LIN {X 0,Y 447.407,Z 741.258,A -85,B 0,C 180,E1 -8717.643,E2 -8717.643} C_VEL
LIN {X 0,Y 446.849,Z 749.798,A -85,B 0,C 180,E1 -8718.663,E2 -8718.663} C_VEL
LIN {X 0,Y 446.393,Z 757.677,A -85,B 0,C 180,E1 -8719.799,E2 -8719.799} C_VEL
LIN {X 0,Y 445.992,Z 765.376,A -85,B 0,C 180,E1 -8721.163,E2 -8721.163} C_VEL
LIN {X 0,Y 445.668,Z 772.472,A -85,B 0,C 180,E1 -8722.753,E2 -8722.753} C_VEL
LIN {X 0,Y 445.494,Z 776.598,A -85,B 0,C 180,E1 -8723.926,E2 -8723.926} C_VEL
LIN {X 0,Y 445.417,Z 780.807,A -85,B 0,C 180,E1 -8725.476,E2 -8725.476} C_VEL
LIN {X 0,Y 445.381,Z 782.67,A -85,B 0,C 180,E1 -8726.382,E2 -8726.382} C_VEL
LIN {X 0,Y 445.433,Z 784.067,A -85,B 0,C 180,E1 -8727.288,E2 -8727.288} C_VEL
LIN {X 0,Y 445.338,Z 785.666,A -85,B 0,C 180,E1 -8729.097,E2 -8729.097} C_VEL
LIN {X 0,Y 445.342,Z 785.882,A -85,B 0,C 180,E1 -8730.001,E2 -8730.001} C_VEL
LIN {X 0,Y 445.338,Z 785.664,A -85,B 0,C 180,E1 -8730.905,E2 -8730.905} C_VEL
LIN {X 0,Y 445.433,Z 784.061,A -85,B 0,C 180,E1 -8732.714,E2 -8732.714} C_VEL
LIN {X 0,Y 445.381,Z 782.661,A -85,B 0,C 180,E1 -8733.62,E2 -8733.62} C_VEL
LIN {X 0,Y 445.482,Z 779.728,A -85,B 0,C 180,E1 -8734.979,E2 -8734.979} C_VEL
LIN {X 0,Y 445.576,Z 774.321,A -85,B 0,C 180,E1 -8736.749,E2 -8736.749} C_VEL
LIN {X 0,Y 445.848,Z 768.627,A -85,B 0,C 180,E1 -8738.157,E2 -8738.157} C_VEL
LIN {X 0,Y 446.16,Z 761.722,A -85,B 0,C 180,E1 -8739.521,E2 -8739.521} C_VEL
LIN {X 0,Y 446.611,Z 753.085,A -85,B 0,C 180,E1 -8740.886,E2 -8740.886} C_VEL
LIN {X 0,Y 447.213,Z 744.233,A -85,B 0,C 180,E1 -8742.019,E2 -8742.019} C_VEL
LIN {X 0,Y 447.682,Z 735.24,A -85,B 0,C 180,E1 -8742.972,E2 -8742.972} C_VEL
LIN {X 0,Y 448.293,Z 723.879,A -85,B 0,C 180,E1 -8743.949,E2 -8743.949} C_VEL
LIN {X 0,Y 448.894,Z 712.012,A -85,B 0,C 180,E1 -8744.74,E2 -8744.74} C_VEL
LIN {X 0,Y 449.496,Z 699.666,A -85,B 0,C 180,E1 -8745.357,E2 -8745.357} C_VEL
LIN {X 0,Y 449.946,Z 686.98,A -85,B 0,C 180,E1 -8745.806,E2 -8745.806} C_VEL
LIN {X 0,Y 450.236,Z 673.706,A -85,B 0,C 180,E1 -8746.086,E2 -8746.086} C_VEL
LIN {X 0,Y 450.721,Z 593.513,A -85,B 0,C 180,E1 -8747.374,E2 -8747.374} C_VEL
LIN {X 0,Y 447.503,Z 573.501,A -85,B 0,C 180,E1 -8747.859,E2 -8747.859} C_VEL
LIN {X 0,Y 448.187,Z 559.557,A -85,B 0,C 180,E1 -8750.421,E2 -8750.421} C_VEL
LIN {X 0,Y 449.049,Z 544.405,A -85,B 0,C 180,E1 -8753.278,E2 -8753.278} C_VEL
LIN {X 0,Y 448.611,Z 539.586,A -85,B 0,C 180,E1 -8754.233,E2 -8754.233} C_VEL
LIN {X 0,Y 446.536,Z 529.051,A -85,B 0,C 180,E1 -8756.444,E2 -8756.444} C_VEL
LIN {X 0,Y 446.452,Z 528.852,A -85,B 0,C 180,E1 -8759.21,E2 -8759.21} C_VEL
LIN {X 0,Y 446.426,Z 528.878,A -85,B 0,C 180,E1 -8762.362,E2 -8762.362} C_VEL
LIN {X 0,Y 446.423,Z 528.875,A -85,B 0,C 180,E1 -8765.626,E2 -8765.626} C_VEL
LIN {X 0,Y 446.448,Z 528.87,A -85,B 0,C 180,E1 -8769.027,E2 -8769.027} C_VEL
LIN {X 0,Y 446.439,Z 528.875,A -85,B 0,C 180,E1 -8772.278,E2 -8772.278} C_VEL
LIN {X 0,Y 446.458,Z 528.871,A -85,B 0,C 180,E1 -8775.104,E2 -8775.104} C_VEL
LIN {X 0,Y 446.432,Z 528.875,A -85,B 0,C 180,E1 -8778.609,E2 -8778.609} C_VEL
LIN {X 0,Y 446.449,Z 528.871,A -85,B 0,C 180,E1 -8780.973,E2 -8780.973} C_VEL
LIN {X 0,Y 446.426,Z 528.877,A -85,B 0,C 180,E1 -8784.374,E2 -8784.374} C_VEL
LIN {X 0,Y 446.426,Z 528.879,A -85,B 0,C 180,E1 -8787.639,E2 -8787.639} C_VEL
LIN {X 0,Y 446.49,Z 528.871,A -85,B 0,C 180,E1 -8791.309,E2 -8791.309} C_VEL
LIN {X 0,Y 446.544,Z 529.135,A -85,B 0,C 180,E1 -8791.774,E2 -8791.774} C_VEL
LIN {X 0,Y 448.876,Z 539.427,A -85,B 0,C 180,E1 -8793.454,E2 -8793.454} C_VEL
LIN {X 0,Y 449.618,Z 544.795,A -85,B 0,C 180,E1 -8794.293,E2 -8794.293} C_VEL
LIN {X 0,Y 448.993,Z 565.446,A -85,B 0,C 180,E1 -8797.299,E2 -8797.299} C_VEL
LIN {X 0,Y 448.285,Z 587.456,A -85,B 0,C 180,E1 -8800.545,E2 -8800.545} C_VEL
LIN {X 0,Y 447.587,Z 611.18,A -85,B 0,C 180,E1 -8804.051,E2 -8804.051} C_VEL
LIN {X 0,Y 446.999,Z 631.561,A -85,B 0,C 180,E1 -8807.047,E2 -8807.047} C_VEL
LIN {X 0,Y 448.391,Z 644.528,A -85,B 0,C 180,E1 -8807.365,E2 -8807.365} C_VEL
LIN {X 0,Y 447.727,Z 703.384,A -85,B 0,C 180,E1 -8808.484,E2 -8808.484} C_VEL
LIN {X 0,Y 447.557,Z 713.56,A -85,B 0,C 180,E1 -8808.823,E2 -8808.823} C_VEL
LIN {X 0,Y 447.25,Z 724.586,A -85,B 0,C 180,E1 -8809.36,E2 -8809.36} C_VEL
LIN {X 0,Y 446.948,Z 734.395,A -85,B 0,C 180,E1 -8810.04,E2 -8810.04} C_VEL
LIN {X 0,Y 446.644,Z 742.148,A -85,B 0,C 180,E1 -8810.719,E2 -8810.719} C_VEL
LIN {X 0,Y 446.274,Z 750.496,A -85,B 0,C 180,E1 -8811.624,E2 -8811.624} C_VEL
LIN {X 0,Y 445.989,Z 758.487,A -85,B 0,C 180,E1 -8812.758,E2 -8812.758} C_VEL
LIN {X 0,Y 445.802,Z 763.618,A -85,B 0,C 180,E1 -8813.664,E2 -8813.664} C_VEL
LIN {X 0,Y 445.686,Z 767.819,A -85,B 0,C 180,E1 -8814.571,E2 -8814.571} C_VEL
LIN {X 0,Y 445.501,Z 771.222,A -85,B 0,C 180,E1 -8815.476,E2 -8815.476} C_VEL
LIN {X 0,Y 445.504,Z 773.912,A -85,B 0,C 180,E1 -8816.382,E2 -8816.382} C_VEL
LIN {X 0,Y 445.455,Z 775.959,A -85,B 0,C 180,E1 -8817.287,E2 -8817.287} C_VEL
LIN {X 0,Y 445.357,Z 777.408,A -85,B 0,C 180,E1 -8818.191,E2 -8818.191} C_VEL
LIN {X 0,Y 445.314,Z 778.286,A -85,B 0,C 180,E1 -8819.096,E2 -8819.096} C_VEL
LIN {X 0,Y 445.315,Z 778.58,A -85,B 0,C 180,E1 -8820,E2 -8820} C_VEL
LIN {X 0,Y 445.315,Z 778.281,A -85,B 0,C 180,E1 -8820.904,E2 -8820.904} C_VEL
LIN {X 0,Y 445.357,Z 777.404,A -85,B 0,C 180,E1 -8821.809,E2 -8821.809} C_VEL
LIN {X 0,Y 445.488,Z 775.061,A -85,B 0,C 180,E1 -8823.165,E2 -8823.165} C_VEL
LIN {X 0,Y 445.477,Z 772.717,A -85,B 0,C 180,E1 -8824.071,E2 -8824.071} C_VEL
LIN {X 0,Y 445.56,Z 769.687,A -85,B 0,C 180,E1 -8824.977,E2 -8824.977} C_VEL
LIN {X 0,Y 445.736,Z 764.784,A -85,B 0,C 180,E1 -8826.11,E2 -8826.11} C_VEL
LIN {X 0,Y 445.92,Z 760.093,A -85,B 0,C 180,E1 -8826.983,E2 -8826.983} C_VEL
LIN {X 0,Y 446.07,Z 753.905,A -85,B 0,C 180,E1 -8827.924,E2 -8827.924} C_VEL
LIN {X 0,Y 446.349,Z 746.57,A -85,B 0,C 180,E1 -8828.831,E2 -8828.831} C_VEL
LIN {X 0,Y 446.748,Z 737.266,A -85,B 0,C 180,E1 -8829.736,E2 -8829.736} C_VEL
LIN {X 0,Y 447.058,Z 728.149,A -85,B 0,C 180,E1 -8830.416,E2 -8830.416} C_VEL
LIN {X 0,Y 447.317,Z 718.258,A -85,B 0,C 180,E1 -8830.982,E2 -8830.982} C_VEL
LIN {X 0,Y 447.568,Z 707.509,A -85,B 0,C 180,E1 -8831.406,E2 -8831.406} C_VEL
LIN {X 0,Y 447.655,Z 697.084,A -85,B 0,C 180,E1 -8831.662,E2 -8831.662} C_VEL
LIN {X 0,Y 448.07,Z 642.126,A -85,B 0,C 180,E1 -8832.648,E2 -8832.648} C_VEL
LIN {X 0,Y 446.85,Z 631.601,A -85,B 0,C 180,E1 -8832.889,E2 -8832.889} C_VEL
LIN {X 0,Y 447.122,Z 621.716,A -85,B 0,C 180,E1 -8834.333,E2 -8834.333} C_VEL
LIN {X 0,Y 447.779,Z 600.173,A -85,B 0,C 180,E1 -8837.586,E2 -8837.586} C_VEL
LIN {X 0,Y 448.48,Z 579.967,A -85,B 0,C 180,E1 -8840.646,E2 -8840.646} C_VEL
LIN {X 0,Y 449.352,Z 556.333,A -85,B 0,C 180,E1 -8844.24,E2 -8844.24} C_VEL
LIN {X 0,Y 449.698,Z 545.085,A -85,B 0,C 180,E1 -8845.95,E2 -8845.95} C_VEL
LIN {X 0,Y 447.465,Z 533.4,A -85,B 0,C 180,E1 -8847.857,E2 -8847.857} C_VEL
LIN {X 0,Y 446.517,Z 528.97,A -85,B 0,C 180,E1 -8848.636,E2 -8848.636} C_VEL
LIN {X 0,Y 446.426,Z 528.879,A -85,B 0,C 180,E1 -8852.361,E2 -8852.361} C_VEL
LIN {X 0,Y 446.426,Z 528.874,A -85,B 0,C 180,E1 -8855.626,E2 -8855.626} C_VEL
LIN {X 0,Y 446.45,Z 528.869,A -85,B 0,C 180,E1 -8859.027,E2 -8859.027} C_VEL
LIN {X 0,Y 446.438,Z 528.854,A -85,B 0,C 180,E1 -8862.277,E2 -8862.277} C_VEL
LIN {X 0,Y 446.46,Z 528.867,A -85,B 0,C 180,E1 -8865.103,E2 -8865.103} C_VEL
LIN {X 0,Y 446.434,Z 528.869,A -85,B 0,C 180,E1 -8868.609,E2 -8868.609} C_VEL
LIN {X 0,Y 446.446,Z 528.861,A -85,B 0,C 180,E1 -8870.973,E2 -8870.973} C_VEL
LIN {X 0,Y 446.424,Z 528.878,A -85,B 0,C 180,E1 -8874.374,E2 -8874.374} C_VEL
LIN {X 0,Y 446.427,Z 528.873,A -85,B 0,C 180,E1 -8877.638,E2 -8877.638} C_VEL
LIN {X 0,Y 446.453,Z 528.873,A -85,B 0,C 180,E1 -8880.79,E2 -8880.79} C_VEL
LIN {X 0,Y 446.483,Z 528.867,A -85,B 0,C 180,E1 -8883.848,E2 -8883.848} C_VEL
LIN {X 0,Y 446.462,Z 528.879,A -85,B 0,C 180,E1 -8887.314,E2 -8887.314} C_VEL
LIN {X 0,Y 446.546,Z 529.43,A -85,B 0,C 180,E1 -8887.563,E2 -8887.563} C_VEL
LIN {X 0,Y 448.137,Z 537.779,A -85,B 0,C 180,E1 -8889.577,E2 -8889.577} C_VEL
LIN {X 0,Y 447.892,Z 544.522,A -85,B 0,C 180,E1 -8891.086,E2 -8891.086} C_VEL
LIN {X 0,Y 447.633,Z 546.914,A -85,B 0,C 180,E1 -8891.469,E2 -8891.469} C_VEL
LIN {X 0,Y 446.932,Z 551.667,A -85,B 0,C 180,E1 -8891.892,E2 -8891.892} C_VEL
LIN {X 0,Y 446.062,Z 557.135,A -85,B 0,C 180,E1 -8892.159,E2 -8892.159} C_VEL
LIN {X 0,Y 444.882,Z 565.287,A -85,B 0,C 180,E1 -8892.361,E2 -8892.361} C_VEL
LIN {X 0,Y 444.177,Z 573.6,A -85,B 0,C 180,E1 -8892.485,E2 -8892.485} C_VEL
LIN {X 0,Y 443.385,Z 657.161,A -85,B 0,C 180,E1 -8893.865,E2 -8893.865} C_VEL
LIN {X 0,Y 443.004,Z 671.025,A -85,B 0,C 180,E1 -8894.294,E2 -8894.294} C_VEL
LIN {X 0,Y 442.518,Z 683.422,A -85,B 0,C 180,E1 -8894.866,E2 -8894.866} C_VEL
LIN {X 0,Y 441.942,Z 695.268,A -85,B 0,C 180,E1 -8895.612,E2 -8895.612} C_VEL
LIN {X 0,Y 441.388,Z 706.67,A -85,B 0,C 180,E1 -8896.537,E2 -8896.537} C_VEL
LIN {X 0,Y 440.763,Z 716.867,A -85,B 0,C 180,E1 -8897.569,E2 -8897.569} C_VEL
LIN {X 0,Y 440.147,Z 726.052,A -85,B 0,C 180,E1 -8898.719,E2 -8898.719} C_VEL
LIN {X 0,Y 439.552,Z 734.97,A -85,B 0,C 180,E1 -8900.102,E2 -8900.102} C_VEL
LIN {X 0,Y 439.104,Z 742.146,A -85,B 0,C 180,E1 -8901.485,E2 -8901.485} C_VEL
LIN {X 0,Y 438.788,Z 746.99,A -85,B 0,C 180,E1 -8902.637,E2 -8902.637} C_VEL
LIN {X 0,Y 438.686,Z 751.69,A -85,B 0,C 180,E1 -8904.022,E2 -8904.022} C_VEL
LIN {X 0,Y 438.424,Z 755.29,A -85,B 0,C 180,E1 -8905.402,E2 -8905.402} C_VEL
LIN {X 0,Y 438.428,Z 757.148,A -85,B 0,C 180,E1 -8906.323,E2 -8906.323} C_VEL
LIN {X 0,Y 438.395,Z 758.551,A -85,B 0,C 180,E1 -8907.243,E2 -8907.243} C_VEL
LIN {X 0,Y 438.255,Z 760.167,A -85,B 0,C 180,E1 -8909.08,E2 -8909.08} C_VEL
LIN {X 0,Y 438.254,Z 760.402,A -85,B 0,C 180,E1 -8909.999,E2 -8909.999} C_VEL
LIN {X 0,Y 438.255,Z 760.216,A -85,B 0,C 180,E1 -8910.918,E2 -8910.918} C_VEL
LIN {X 0,Y 438.392,Z 758.667,A -85,B 0,C 180,E1 -8912.756,E2 -8912.756} C_VEL
LIN {X 0,Y 438.413,Z 757.314,A -85,B 0,C 180,E1 -8913.676,E2 -8913.676} C_VEL
LIN {X 0,Y 438.481,Z 754.45,A -85,B 0,C 180,E1 -8915.057,E2 -8915.057} C_VEL
LIN {X 0,Y 438.693,Z 750.563,A -85,B 0,C 180,E1 -8916.438,E2 -8916.438} C_VEL
LIN {X 0,Y 438.902,Z 745.555,A -85,B 0,C 180,E1 -8917.822,E2 -8917.822} C_VEL
LIN {X 0,Y 439.321,Z 739.248,A -85,B 0,C 180,E1 -8919.204,E2 -8919.204} C_VEL
LIN {X 0,Y 439.803,Z 731.349,A -85,B 0,C 180,E1 -8920.588,E2 -8920.588} C_VEL
LIN {X 0,Y 440.285,Z 723.299,A -85,B 0,C 180,E1 -8921.742,E2 -8921.742} C_VEL
LIN {X 0,Y 441.015,Z 713.467,A -85,B 0,C 180,E1 -8922.89,E2 -8922.89} C_VEL
LIN {X 0,Y 441.544,Z 702.694,A -85,B 0,C 180,E1 -8923.907,E2 -8923.907} C_VEL
LIN {X 0,Y 442.142,Z 691.584,A -85,B 0,C 180,E1 -8924.733,E2 -8924.733} C_VEL
LIN {X 0,Y 442.72,Z 679.605,A -85,B 0,C 180,E1 -8925.419,E2 -8925.419} C_VEL
LIN {X 0,Y 443.147,Z 666.472,A -85,B 0,C 180,E1 -8925.965,E2 -8925.965} C_VEL
LIN {X 0,Y 443.508,Z 653.263,A -85,B 0,C 180,E1 -8926.306,E2 -8926.306} C_VEL
LIN {X 0,Y 444.113,Z 567.024,A -85,B 0,C 180,E1 -8927.72,E2 -8927.72} C_VEL
LIN {X 0,Y 440.768,Z 550.156,A -85,B 0,C 180,E1 -8928.171,E2 -8928.171} C_VEL
LIN {X 0,Y 440.78,Z 547.921,A -85,B 0,C 180,E1 -8928.595,E2 -8928.595} C_VEL
LIN {X 0,Y 441.2,Z 539.437,A -85,B 0,C 180,E1 -8930.513,E2 -8930.513} C_VEL
LIN {X 0,Y 439.437,Z 529.822,A -85,B 0,C 180,E1 -8932.912,E2 -8932.912} C_VEL
LIN {X 0,Y 439.433,Z 529.742,A -85,B 0,C 180,E1 -8936.41,E2 -8936.41} C_VEL
LIN {X 0,Y 439.416,Z 529.744,A -85,B 0,C 180,E1 -8938.672,E2 -8938.672} C_VEL
LIN {X 0,Y 439.369,Z 529.753,A -85,B 0,C 180,E1 -8942.03,E2 -8942.03} C_VEL
LIN {X 0,Y 439.394,Z 529.752,A -85,B 0,C 180,E1 -8945.34,E2 -8945.34} C_VEL
LIN {X 0,Y 439.387,Z 529.75,A -85,B 0,C 180,E1 -8948.593,E2 -8948.593} C_VEL
LIN {X 0,Y 439.386,Z 529.751,A -85,B 0,C 180,E1 -8951.256,E2 -8951.256} C_VEL
LIN {X 0,Y 439.401,Z 529.741,A -85,B 0,C 180,E1 -8954.728,E2 -8954.728} C_VEL
LIN {X 0,Y 439.392,Z 529.752,A -85,B 0,C 180,E1 -8957.795,E2 -8957.795} C_VEL
LIN {X 0,Y 439.447,Z 529.734,A -85,B 0,C 180,E1 -8960.229,E2 -8960.229} C_VEL
LIN {X 0,Y 439.373,Z 529.756,A -85,B 0,C 180,E1 -8963.712,E2 -8963.712} C_VEL
LIN {X 0,Y 439.367,Z 529.754,A -85,B 0,C 180,E1 -8967.053,E2 -8967.053} C_VEL
LIN {X 0,Y 439.39,Z 529.749,A -85,B 0,C 180,E1 -8970.275,E2 -8970.275} C_VEL
LIN {X 0,Y 439.427,Z 529.748,A -85,B 0,C 180,E1 -8973.588,E2 -8973.588} C_VEL
LIN {X 0,Y 439.38,Z 529.748,A -85,B 0,C 180,E1 -8976.429,E2 -8976.429} C_VEL
LIN {X 0,Y 439.382,Z 529.752,A -85,B 0,C 180,E1 -8979.397,E2 -8979.397} C_VEL
LIN {X 0,Y 439.424,Z 529.741,A -85,B 0,C 180,E1 -8982.309,E2 -8982.309} C_VEL
LIN {X 0,Y 439.44,Z 529.741,A -85,B 0,C 180,E1 -8985.174,E2 -8985.174} C_VEL
LIN {X 0,Y 439.476,Z 529.738,A -85,B 0,C 180,E1 -8988.001,E2 -8988.001} C_VEL
LIN {X 0,Y 439.54,Z 529.734,A -85,B 0,C 180,E1 -8991.726,E2 -8991.726} C_VEL
LIN {X 0,Y 439.614,Z 529.72,A -85,B 0,C 180,E1 -8994.496,E2 -8994.496} C_VEL
LIN {X 0,Y 439.628,Z 529.718,A -85,B 0,C 180,E1 -8998.168,E2 -8998.168} C_VEL
LIN {X 0,Y 439.757,Z 529.706,A -85,B 0,C 180,E1 -9000,E2 -9000} C_VEL
LIN {X 0,Y 439.649,Z 529.712,A -85,B 0,C 180,E1 -9002.749,E2 -9002.749} C_VEL
LIN {X 0,Y 439.61,Z 529.721,A -85,B 0,C 180,E1 -9006.425,E2 -9006.425} C_VEL
LIN {X 0,Y 439.493,Z 529.737,A -85,B 0,C 180,E1 -9009.202,E2 -9009.202} C_VEL
LIN {X 0,Y 439.496,Z 529.735,A -85,B 0,C 180,E1 -9012.727,E2 -9012.727} C_VEL
LIN {X 0,Y 439.44,Z 529.737,A -85,B 0,C 180,E1 -9016.349,E2 -9016.349} C_VEL
LIN {X 0,Y 439.423,Z 529.751,A -85,B 0,C 180,E1 -9019.625,E2 -9019.625} C_VEL
LIN {X 0,Y 439.358,Z 529.75,A -85,B 0,C 180,E1 -9022.576,E2 -9022.576} C_VEL
LIN {X 0,Y 439.399,Z 529.752,A -85,B 0,C 180,E1 -9025.585,E2 -9025.585} C_VEL
LIN {X 0,Y 439.411,Z 529.747,A -85,B 0,C 180,E1 -9028.674,E2 -9028.674} C_VEL
LIN {X 0,Y 439.375,Z 529.754,A -85,B 0,C 180,E1 -9032.034,E2 -9032.034} C_VEL
LIN {X 0,Y 439.39,Z 529.748,A -85,B 0,C 180,E1 -9035.342,E2 -9035.342} C_VEL
LIN {X 0,Y 439.385,Z 529.749,A -85,B 0,C 180,E1 -9038.595,E2 -9038.595} C_VEL
LIN {X 0,Y 439.383,Z 529.752,A -85,B 0,C 180,E1 -9041.258,E2 -9041.258} C_VEL
LIN {X 0,Y 439.4,Z 529.748,A -85,B 0,C 180,E1 -9044.73,E2 -9044.73} C_VEL
LIN {X 0,Y 439.408,Z 529.749,A -85,B 0,C 180,E1 -9047.799,E2 -9047.799} C_VEL
LIN {X 0,Y 439.447,Z 529.739,A -85,B 0,C 180,E1 -9050.231,E2 -9050.231} C_VEL
LIN {X 0,Y 439.374,Z 529.748,A -85,B 0,C 180,E1 -9053.714,E2 -9053.714} C_VEL
LIN {X 0,Y 439.37,Z 529.733,A -85,B 0,C 180,E1 -9057.055,E2 -9057.055} C_VEL
LIN {X 0,Y 439.38,Z 529.723,A -85,B 0,C 180,E1 -9060.275,E2 -9060.275} C_VEL
LIN {X 0,Y 439.469,Z 529.836,A -85,B 0,C 180,E1 -9063.272,E2 -9063.272} C_VEL
LIN {X 0,Y 441.813,Z 541.718,A -85,B 0,C 180,E1 -9065.821,E2 -9065.821} C_VEL
LIN {X 0,Y 442.142,Z 545.523,A -85,B 0,C 180,E1 -9066.586,E2 -9066.586} C_VEL
LIN {X 0,Y 441.101,Z 562.606,A -85,B 0,C 180,E1 -9069.856,E2 -9069.856} C_VEL
LIN {X 0,Y 440.59,Z 573.22,A -85,B 0,C 180,E1 -9071.841,E2 -9071.841} C_VEL
LIN {X 0,Y 442.189,Z 582.98,A -85,B 0,C 180,E1 -9072.105,E2 -9072.105} C_VEL
LIN {X 0,Y 444.109,Z 596.392,A -85,B 0,C 180,E1 -9072.407,E2 -9072.407} C_VEL
LIN {X 0,Y 443.294,Z 681.341,A -85,B 0,C 180,E1 -9073.805,E2 -9073.805} C_VEL
LIN {X 0,Y 442.826,Z 694.585,A -85,B 0,C 180,E1 -9074.201,E2 -9074.201} C_VEL
LIN {X 0,Y 442.286,Z 707.863,A -85,B 0,C 180,E1 -9074.801,E2 -9074.801} C_VEL
LIN {X 0,Y 441.659,Z 719.016,A -85,B 0,C 180,E1 -9075.486,E2 -9075.486} C_VEL
LIN {X 0,Y 441.048,Z 729.687,A -85,B 0,C 180,E1 -9076.323,E2 -9076.323} C_VEL
LIN {X 0,Y 440.443,Z 741.055,A -85,B 0,C 180,E1 -9077.444,E2 -9077.444} C_VEL
LIN {X 0,Y 439.873,Z 749.594,A -85,B 0,C 180,E1 -9078.481,E2 -9078.481} C_VEL
LIN {X 0,Y 439.371,Z 757.473,A -85,B 0,C 180,E1 -9079.634,E2 -9079.634} C_VEL
LIN {X 0,Y 438.937,Z 765.171,A -85,B 0,C 180,E1 -9081.02,E2 -9081.02} C_VEL
LIN {X 0,Y 438.606,Z 772.267,A -85,B 0,C 180,E1 -9082.636,E2 -9082.636} C_VEL
LIN {X 0,Y 438.393,Z 776.825,A -85,B 0,C 180,E1 -9083.967,E2 -9083.967} C_VEL
LIN {X 0,Y 438.346,Z 780.603,A -85,B 0,C 180,E1 -9085.403,E2 -9085.403} C_VEL
LIN {X 0,Y 438.283,Z 782.465,A -85,B 0,C 180,E1 -9086.323,E2 -9086.323} C_VEL
LIN {X 0,Y 438.341,Z 783.863,A -85,B 0,C 180,E1 -9087.244,E2 -9087.244} C_VEL
LIN {X 0,Y 438.252,Z 785.462,A -85,B 0,C 180,E1 -9089.082,E2 -9089.082} C_VEL
LIN {X 0,Y 438.253,Z 785.678,A -85,B 0,C 180,E1 -9090.001,E2 -9090.001} C_VEL
LIN {X 0,Y 438.278,Z 784.851,A -85,B 0,C 180,E1 -9091.839,E2 -9091.839} C_VEL
LIN {X 0,Y 438.341,Z 783.856,A -85,B 0,C 180,E1 -9092.758,E2 -9092.758} C_VEL
LIN {X 0,Y 438.283,Z 782.456,A -85,B 0,C 180,E1 -9093.678,E2 -9093.678} C_VEL
LIN {X 0,Y 438.392,Z 779.522,A -85,B 0,C 180,E1 -9095.059,E2 -9095.059} C_VEL
LIN {X 0,Y 438.449,Z 775.547,A -85,B 0,C 180,E1 -9096.443,E2 -9096.443} C_VEL
LIN {X 0,Y 438.724,Z 769.432,A -85,B 0,C 180,E1 -9098.058,E2 -9098.058} C_VEL
LIN {X 0,Y 439.066,Z 762.753,A -85,B 0,C 180,E1 -9099.444,E2 -9099.444} C_VEL
LIN {X 0,Y 439.523,Z 754.466,A -85,B 0,C 180,E1 -9100.83,E2 -9100.83} C_VEL
LIN {X 0,Y 440.111,Z 745.976,A -85,B 0,C 180,E1 -9101.982,E2 -9101.982} C_VEL
LIN {X 0,Y 440.68,Z 735.869,A -85,B 0,C 180,E1 -9103.098,E2 -9103.098} C_VEL
LIN {X 0,Y 441.296,Z 725.1,A -85,B 0,C 180,E1 -9104.057,E2 -9104.057} C_VEL
LIN {X 0,Y 441.923,Z 713.727,A -85,B 0,C 180,E1 -9104.86,E2 -9104.86} C_VEL
LIN {X 0,Y 442.547,Z 702.06,A -85,B 0,C 180,E1 -9105.486,E2 -9105.486} C_VEL
LIN {X 0,Y 443.011,Z 689.516,A -85,B 0,C 180,E1 -9105.971,E2 -9105.971} C_VEL
LIN {X 0,Y 443.385,Z 676.797,A -85,B 0,C 180,E1 -9106.282,E2 -9106.282} C_VEL
LIN {X 0,Y 443.999,Z 594.924,A -85,B 0,C 180,E1 -9107.619,E2 -9107.619} C_VEL
LIN {X 0,Y 440.562,Z 573.533,A -85,B 0,C 180,E1 -9108.133,E2 -9108.133} C_VEL
LIN {X 0,Y 440.689,Z 570.679,A -85,B 0,C 180,E1 -9108.6,E2 -9108.6} C_VEL
LIN {X 0,Y 441.86,Z 550.549,A -85,B 0,C 180,E1 -9112.442,E2 -9112.442} C_VEL
LIN {X 0,Y 442.138,Z 544.222,A -85,B 0,C 180,E1 -9113.664,E2 -9113.664} C_VEL
LIN {X 0,Y 440.34,Z 534.062,A -85,B 0,C 180,E1 -9115.777,E2 -9115.777} C_VEL
LIN {X 0,Y 439.475,Z 529.804,A -85,B 0,C 180,E1 -9116.746,E2 -9116.746} C_VEL
LIN {X 0,Y 439.385,Z 529.736,A -85,B 0,C 180,E1 -9119.726,E2 -9119.726} C_VEL
LIN {X 0,Y 439.376,Z 529.754,A -85,B 0,C 180,E1 -9122.946,E2 -9122.946} C_VEL
LIN {X 0,Y 439.378,Z 529.756,A -85,B 0,C 180,E1 -9126.288,E2 -9126.288} C_VEL
LIN {X 0,Y 439.405,Z 529.753,A -85,B 0,C 180,E1 -9129.849,E2 -9129.849} C_VEL
LIN {X 0,Y 439.386,Z 529.752,A -85,B 0,C 180,E1 -9132.627,E2 -9132.627} C_VEL
LIN {X 0,Y 439.405,Z 529.75,A -85,B 0,C 180,E1 -9135.271,E2 -9135.271} C_VEL
LIN {X 0,Y 439.392,Z 529.752,A -85,B 0,C 180,E1 -9138.743,E2 -9138.743} C_VEL
LIN {X 0,Y 439.386,Z 529.755,A -85,B 0,C 180,E1 -9141.607,E2 -9141.607} C_VEL
LIN {X 0,Y 439.405,Z 529.749,A -85,B 0,C 180,E1 -9144.844,E2 -9144.844} C_VEL
LIN {X 0,Y 439.377,Z 529.758,A -85,B 0,C 180,E1 -9148.14,E2 -9148.14} C_VEL
LIN {X 0,Y 439.479,Z 529.934,A -85,B 0,C 180,E1 -9151.397,E2 -9151.397} C_VEL
LIN {X 0,Y 442.015,Z 540.745,A -85,B 0,C 180,E1 -9153.218,E2 -9153.218} C_VEL
LIN {X 0,Y 442.837,Z 546.431,A -85,B 0,C 180,E1 -9154.123,E2 -9154.123} C_VEL
LIN {X 0,Y 442.172,Z 565.852,A -85,B 0,C 180,E1 -9156.992,E2 -9156.992} C_VEL
LIN {X 0,Y 441.413,Z 587.891,A -85,B 0,C 180,E1 -9160.283,E2 -9160.283} C_VEL
LIN {X 0,Y 440.69,Z 611.421,A -85,B 0,C 180,E1 -9163.794,E2 -9163.794} C_VEL
LIN {X 0,Y 440.074,Z 631.467,A -85,B 0,C 180,E1 -9166.782,E2 -9166.782} C_VEL
LIN {X 0,Y 441.551,Z 645.299,A -85,B 0,C 180,E1 -9167.145,E2 -9167.145} C_VEL
LIN {X 0,Y 440.795,Z 704.212,A -85,B 0,C 180,E1 -9168.3,E2 -9168.3} C_VEL
LIN {X 0,Y 440.605,Z 713.419,A -85,B 0,C 180,E1 -9168.616,E2 -9168.616} C_VEL
LIN {X 0,Y 440.309,Z 723.945,A -85,B 0,C 180,E1 -9169.132,E2 -9169.132} C_VEL
LIN {X 0,Y 439.986,Z 733.226,A -85,B 0,C 180,E1 -9169.764,E2 -9169.764} C_VEL
LIN {X 0,Y 439.677,Z 741.161,A -85,B 0,C 180,E1 -9170.454,E2 -9170.454} C_VEL
LIN {X 0,Y 439.334,Z 748.677,A -85,B 0,C 180,E1 -9171.259,E2 -9171.259} C_VEL
LIN {X 0,Y 439.039,Z 755.676,A -85,B 0,C 180,E1 -9172.18,E2 -9172.18} C_VEL
LIN {X 0,Y 438.831,Z 761.873,A -85,B 0,C 180,E1 -9173.194,E2 -9173.194} C_VEL
LIN {X 0,Y 438.731,Z 766.011,A -85,B 0,C 180,E1 -9174.023,E2 -9174.023} C_VEL
LIN {X 0,Y 438.517,Z 769.796,A -85,B 0,C 180,E1 -9174.943,E2 -9174.943} C_VEL
LIN {X 0,Y 438.435,Z 772.823,A -85,B 0,C 180,E1 -9175.863,E2 -9175.863} C_VEL
LIN {X 0,Y 438.388,Z 776.047,A -85,B 0,C 180,E1 -9177.243,E2 -9177.243} C_VEL
LIN {X 0,Y 438.28,Z 777.486,A -85,B 0,C 180,E1 -9178.162,E2 -9178.162} C_VEL
LIN {X 0,Y 438.229,Z 778.351,A -85,B 0,C 180,E1 -9179.081,E2 -9179.081} C_VEL
LIN {X 0,Y 438.227,Z 778.636,A -85,B 0,C 180,E1 -9180,E2 -9180} C_VEL
LIN {X 0,Y 438.23,Z 778.324,A -85,B 0,C 180,E1 -9180.919,E2 -9180.919} C_VEL
LIN {X 0,Y 438.28,Z 777.425,A -85,B 0,C 180,E1 -9181.838,E2 -9181.838} C_VEL
LIN {X 0,Y 438.415,Z 775.03,A -85,B 0,C 180,E1 -9183.216,E2 -9183.216} C_VEL
LIN {X 0,Y 438.413,Z 771.156,A -85,B 0,C 180,E1 -9184.597,E2 -9184.597} C_VEL
LIN {X 0,Y 438.566,Z 767.72,A -85,B 0,C 180,E1 -9185.518,E2 -9185.518} C_VEL
LIN {X 0,Y 438.729,Z 762.194,A -85,B 0,C 180,E1 -9186.693,E2 -9186.693} C_VEL
LIN {X 0,Y 438.954,Z 755.305,A -85,B 0,C 180,E1 -9187.822,E2 -9187.822} C_VEL
LIN {X 0,Y 439.244,Z 748.216,A -85,B 0,C 180,E1 -9188.743,E2 -9188.743} C_VEL
LIN {X 0,Y 439.644,Z 739.42,A -85,B 0,C 180,E1 -9189.663,E2 -9189.663} C_VEL
LIN {X 0,Y 439.996,Z 729.246,A -85,B 0,C 180,E1 -9190.468,E2 -9190.468} C_VEL
LIN {X 0,Y 440.26,Z 719.62,A -85,B 0,C 180,E1 -9191.044,E2 -9191.044} C_VEL
LIN {X 0,Y 440.558,Z 708.014,A -85,B 0,C 180,E1 -9191.531,E2 -9191.531} C_VEL
LIN {X 0,Y 440.661,Z 696.322,A -85,B 0,C 180,E1 -9191.82,E2 -9191.82} C_VEL
LIN {X 0,Y 441.144,Z 643.139,A -85,B 0,C 180,E1 -9192.802,E2 -9192.802} C_VEL
LIN {X 0,Y 439.846,Z 631.675,A -85,B 0,C 180,E1 -9193.069,E2 -9193.069} C_VEL
LIN {X 0,Y 439.905,Z 627.77,A -85,B 0,C 180,E1 -9193.61,E2 -9193.61} C_VEL
LIN {X 0,Y 440.584,Z 606.554,A -85,B 0,C 180,E1 -9196.843,E2 -9196.843} C_VEL
LIN {X 0,Y 441.414,Z 583.613,A -85,B 0,C 180,E1 -9200.347,E2 -9200.347} C_VEL
LIN {X 0,Y 442.329,Z 560.418,A -85,B 0,C 180,E1 -9203.901,E2 -9203.901} C_VEL
LIN {X 0,Y 442.852,Z 547.573,A -85,B 0,C 180,E1 -9205.876,E2 -9205.876} C_VEL
LIN {X 0,Y 441.331,Z 538.658,A -85,B 0,C 180,E1 -9207.333,E2 -9207.333} C_VEL
LIN {X 0,Y 439.473,Z 529.86,A -85,B 0,C 180,E1 -9208.833,E2 -9208.833} C_VEL
LIN {X 0,Y 439.374,Z 529.756,A -85,B 0,C 180,E1 -9212.03,E2 -9212.03} C_VEL
LIN {X 0,Y 439.401,Z 529.749,A -85,B 0,C 180,E1 -9215.341,E2 -9215.341} C_VEL
LIN {X 0,Y 439.388,Z 529.754,A -85,B 0,C 180,E1 -9218.595,E2 -9218.595} C_VEL
LIN {X 0,Y 439.393,Z 529.735,A -85,B 0,C 180,E1 -9221.257,E2 -9221.257} C_VEL
LIN {X 0,Y 439.406,Z 529.741,A -85,B 0,C 180,E1 -9224.729,E2 -9224.729} C_VEL
LIN {X 0,Y 439.403,Z 529.748,A -85,B 0,C 180,E1 -9227.796,E2 -9227.796} C_VEL
LIN {X 0,Y 439.415,Z 529.734,A -85,B 0,C 180,E1 -9230.225,E2 -9230.225} C_VEL
LIN {X 0,Y 439.378,Z 529.752,A -85,B 0,C 180,E1 -9233.713,E2 -9233.713} C_VEL
LIN {X 0,Y 439.377,Z 529.754,A -85,B 0,C 180,E1 -9237.054,E2 -9237.054} C_VEL
LIN {X 0,Y 439.387,Z 529.754,A -85,B 0,C 180,E1 -9240.274,E2 -9240.274} C_VEL
LIN {X 0,Y 439.432,Z 529.745,A -85,B 0,C 180,E1 -9243.396,E2 -9243.396} C_VEL
LIN {X 0,Y 439.423,Z 529.751,A -85,B 0,C 180,E1 -9246.93,E2 -9246.93} C_VEL
LIN {X 0,Y 439.493,Z 530.134,A -85,B 0,C 180,E1 -9247.307,E2 -9247.307} C_VEL
LIN {X 0,Y 441.174,Z 539.02,A -85,B 0,C 180,E1 -9249.484,E2 -9249.484} C_VEL
LIN {X 0,Y 440.75,Z 549.9,A -85,B 0,C 180,E1 -9251.899,E2 -9251.899} C_VEL
LIN {X 0,Y 441.535,Z 554.074,A -85,B 0,C 180,E1 -9252.048,E2 -9252.048} C_VEL
LIN {X 0,Y 444.252,Z 568.242,A -85,B 0,C 180,E1 -9252.399,E2 -9252.399} C_VEL
LIN {X 0,Y 444.177,Z 573.6,A -85,B 0,C 180,E1 -9252.485,E2 -9252.485} C_VEL
LIN {X 0,Y 443.413,Z 579.441,A -85,B 0,C 180,E1 -9252.551,E2 -9252.551} C_VEL
LIN {X 0,Y 437.959,Z 598.476,A -85,B 0,C 180,E1 -9252.644,E2 -9252.644} C_VEL
LIN {X 0,Y 437.216,Z 604.316,A -85,B 0,C 180,E1 -9252.712,E2 -9252.712} C_VEL
LIN {X 0,Y 436.591,Z 657.383,A -85,B 0,C 180,E1 -9253.607,E2 -9253.607} C_VEL
LIN {X 0,Y 436.186,Z 671.241,A -85,B 0,C 180,E1 -9254.042,E2 -9254.042} C_VEL
LIN {X 0,Y 435.679,Z 683.635,A -85,B 0,C 180,E1 -9254.623,E2 -9254.623} C_VEL
LIN {X 0,Y 435.064,Z 695.479,A -85,B 0,C 180,E1 -9255.38,E2 -9255.38} C_VEL
LIN {X 0,Y 434.474,Z 707.332,A -85,B 0,C 180,E1 -9256.361,E2 -9256.361} C_VEL
LIN {X 0,Y 433.842,Z 717.076,A -85,B 0,C 180,E1 -9257.367,E2 -9257.367} C_VEL
LIN {X 0,Y 433.184,Z 726.26,A -85,B 0,C 180,E1 -9258.536,E2 -9258.536} C_VEL
LIN {X 0,Y 432.557,Z 735.177,A -85,B 0,C 180,E1 -9259.94,E2 -9259.94} C_VEL
LIN {X 0,Y 432.091,Z 742.353,A -85,B 0,C 180,E1 -9261.346,E2 -9261.346} C_VEL
LIN {X 0,Y 431.736,Z 747.197,A -85,B 0,C 180,E1 -9262.516,E2 -9262.516} C_VEL
LIN {X 0,Y 431.617,Z 751.896,A -85,B 0,C 180,E1 -9263.924,E2 -9263.924} C_VEL
LIN {X 0,Y 431.352,Z 755.496,A -85,B 0,C 180,E1 -9265.326,E2 -9265.326} C_VEL
LIN {X 0,Y 431.333,Z 757.354,A -85,B 0,C 180,E1 -9266.262,E2 -9266.262} C_VEL
LIN {X 0,Y 431.326,Z 758.755,A -85,B 0,C 180,E1 -9267.197,E2 -9267.197} C_VEL
LIN {X 0,Y 431.172,Z 760.372,A -85,B 0,C 180,E1 -9269.065,E2 -9269.065} C_VEL
LIN {X 0,Y 431.168,Z 760.607,A -85,B 0,C 180,E1 -9269.999,E2 -9269.999} C_VEL
LIN {X 0,Y 431.172,Z 760.42,A -85,B 0,C 180,E1 -9270.933,E2 -9270.933} C_VEL
LIN {X 0,Y 431.324,Z 758.871,A -85,B 0,C 180,E1 -9272.801,E2 -9272.801} C_VEL
LIN {X 0,Y 431.318,Z 757.518,A -85,B 0,C 180,E1 -9273.736,E2 -9273.736} C_VEL
LIN {X 0,Y 431.427,Z 754.653,A -85,B 0,C 180,E1 -9275.139,E2 -9275.139} C_VEL
LIN {X 0,Y 431.64,Z 750.344,A -85,B 0,C 180,E1 -9276.68,E2 -9276.68} C_VEL
LIN {X 0,Y 431.871,Z 745.758,A -85,B 0,C 180,E1 -9277.95,E2 -9277.95} C_VEL
LIN {X 0,Y 432.311,Z 739.45,A -85,B 0,C 180,E1 -9279.355,E2 -9279.355} C_VEL
LIN {X 0,Y 432.839,Z 731.551,A -85,B 0,C 180,E1 -9280.761,E2 -9280.761} C_VEL
LIN {X 0,Y 433.323,Z 723.501,A -85,B 0,C 180,E1 -9281.933,E2 -9281.933} C_VEL
LIN {X 0,Y 434.091,Z 713.668,A -85,B 0,C 180,E1 -9283.1,E2 -9283.1} C_VEL
LIN {X 0,Y 434.674,Z 702.622,A -85,B 0,C 180,E1 -9284.154,E2 -9284.154} C_VEL
LIN {X 0,Y 435.303,Z 691.781,A -85,B 0,C 180,E1 -9284.969,E2 -9284.969} C_VEL
LIN {X 0,Y 435.903,Z 679.8,A -85,B 0,C 180,E1 -9285.667,E2 -9285.667} C_VEL
LIN {X 0,Y 436.329,Z 667.541,A -85,B 0,C 180,E1 -9286.191,E2 -9286.191} C_VEL
LIN {X 0,Y 436.672,Z 654.948,A -85,B 0,C 180,E1 -9286.538,E2 -9286.538} C_VEL
LIN {X 0,Y 437.389,Z 568.131,A -85,B 0,C 180,E1 -9287.986,E2 -9287.986} C_VEL
LIN {X 0,Y 433.874,Z 550.521,A -85,B 0,C 180,E1 -9288.461,E2 -9288.461} C_VEL
LIN {X 0,Y 433.83,Z 549.071,A -85,B 0,C 180,E1 -9288.683,E2 -9288.683} C_VEL
LIN {X 0,Y 434.243,Z 541.496,A -85,B 0,C 180,E1 -9290.419,E2 -9290.419} C_VEL
LIN {X 0,Y 432.851,Z 532.983,A -85,B 0,C 180,E1 -9292.511,E2 -9292.511} C_VEL
LIN {X 0,Y 432.397,Z 530.646,A -85,B 0,C 180,E1 -9293.18,E2 -9293.18} C_VEL
LIN {X 0,Y 432.399,Z 530.618,A -85,B 0,C 180,E1 -9296.626,E2 -9296.626} C_VEL
LIN {X 0,Y 432.342,Z 530.621,A -85,B 0,C 180,E1 -9299.186,E2 -9299.186} C_VEL
LIN {X 0,Y 432.321,Z 530.63,A -85,B 0,C 180,E1 -9302.442,E2 -9302.442} C_VEL
LIN {X 0,Y 432.343,Z 530.627,A -85,B 0,C 180,E1 -9305.631,E2 -9305.631} C_VEL
LIN {X 0,Y 432.35,Z 530.627,A -85,B 0,C 180,E1 -9308.715,E2 -9308.715} C_VEL
LIN {X 0,Y 432.332,Z 530.632,A -85,B 0,C 180,E1 -9311.796,E2 -9311.796} C_VEL
LIN {X 0,Y 432.336,Z 530.62,A -85,B 0,C 180,E1 -9314.345,E2 -9314.345} C_VEL
LIN {X 0,Y 432.316,Z 530.63,A -85,B 0,C 180,E1 -9317.015,E2 -9317.015} C_VEL
LIN {X 0,Y 432.352,Z 530.62,A -85,B 0,C 180,E1 -9319.816,E2 -9319.816} C_VEL
LIN {X 0,Y 432.312,Z 530.624,A -85,B 0,C 180,E1 -9323.022,E2 -9323.022} C_VEL
LIN {X 0,Y 432.357,Z 530.626,A -85,B 0,C 180,E1 -9325.995,E2 -9325.995} C_VEL
LIN {X 0,Y 432.389,Z 530.625,A -85,B 0,C 180,E1 -9329.743,E2 -9329.743} C_VEL
LIN {X 0,Y 432.394,Z 530.621,A -85,B 0,C 180,E1 -9333.372,E2 -9333.372} C_VEL
LIN {X 0,Y 432.364,Z 530.624,A -85,B 0,C 180,E1 -9336.023,E2 -9336.023} C_VEL
LIN {X 0,Y 432.343,Z 530.624,A -85,B 0,C 180,E1 -9339.046,E2 -9339.046} C_VEL
LIN {X 0,Y 432.371,Z 530.622,A -85,B 0,C 180,E1 -9342.011,E2 -9342.011} C_VEL
LIN {X 0,Y 432.388,Z 530.617,A -85,B 0,C 180,E1 -9344.926,E2 -9344.926} C_VEL
LIN {X 0,Y 432.451,Z 530.615,A -85,B 0,C 180,E1 -9347.803,E2 -9347.803} C_VEL
LIN {X 0,Y 432.484,Z 530.61,A -85,B 0,C 180,E1 -9351.59,E2 -9351.59} C_VEL
LIN {X 0,Y 432.591,Z 530.595,A -85,B 0,C 180,E1 -9354.406,E2 -9354.406} C_VEL
LIN {X 0,Y 432.598,Z 530.594,A -85,B 0,C 180,E1 -9358.138,E2 -9358.138} C_VEL
LIN {X 0,Y 432.727,Z 530.581,A -85,B 0,C 180,E1 -9360,E2 -9360} C_VEL
LIN {X 0,Y 432.599,Z 530.591,A -85,B 0,C 180,E1 -9362.794,E2 -9362.794} C_VEL
LIN {X 0,Y 432.565,Z 530.599,A -85,B 0,C 180,E1 -9366.53,E2 -9366.53} C_VEL
LIN {X 0,Y 432.436,Z 530.616,A -85,B 0,C 180,E1 -9369.353,E2 -9369.353} C_VEL
LIN {X 0,Y 432.437,Z 530.615,A -85,B 0,C 180,E1 -9372.812,E2 -9372.812} C_VEL
LIN {X 0,Y 432.405,Z 530.613,A -85,B 0,C 180,E1 -9376.479,E2 -9376.479} C_VEL
LIN {X 0,Y 432.366,Z 530.625,A -85,B 0,C 180,E1 -9379.959,E2 -9379.959} C_VEL
LIN {X 0,Y 432.312,Z 530.629,A -85,B 0,C 180,E1 -9382.965,E2 -9382.965} C_VEL
LIN {X 0,Y 432.358,Z 530.622,A -85,B 0,C 180,E1 -9386.033,E2 -9386.033} C_VEL
LIN {X 0,Y 432.336,Z 530.63,A -85,B 0,C 180,E1 -9389.188,E2 -9389.188} C_VEL
LIN {X 0,Y 432.321,Z 530.63,A -85,B 0,C 180,E1 -9392.443,E2 -9392.443} C_VEL
LIN {X 0,Y 432.34,Z 530.621,A -85,B 0,C 180,E1 -9395.633,E2 -9395.633} C_VEL
LIN {X 0,Y 432.347,Z 530.625,A -85,B 0,C 180,E1 -9398.717,E2 -9398.717} C_VEL
LIN {X 0,Y 432.328,Z 530.625,A -85,B 0,C 180,E1 -9401.798,E2 -9401.798} C_VEL
LIN {X 0,Y 432.374,Z 530.627,A -85,B 0,C 180,E1 -9405.659,E2 -9405.659} C_VEL
LIN {X 0,Y 432.369,Z 530.625,A -85,B 0,C 180,E1 -9408.393,E2 -9408.393} C_VEL
LIN {X 0,Y 432.349,Z 530.612,A -85,B 0,C 180,E1 -9411.853,E2 -9411.853} C_VEL
LIN {X 0,Y 432.338,Z 530.633,A -85,B 0,C 180,E1 -9415.324,E2 -9415.324} C_VEL
LIN {X 0,Y 432.319,Z 530.584,A -85,B 0,C 180,E1 -9418.655,E2 -9418.655} C_VEL
LIN {X 0,Y 432.382,Z 530.626,A -85,B 0,C 180,E1 -9421.878,E2 -9421.878} C_VEL
LIN {X 0,Y 432.429,Z 530.806,A -85,B 0,C 180,E1 -9423.06,E2 -9423.06} C_VEL
LIN {X 0,Y 434.818,Z 542.801,A -85,B 0,C 180,E1 -9425.661,E2 -9425.661} C_VEL
LIN {X 0,Y 435.207,Z 546.733,A -85,B 0,C 180,E1 -9426.468,E2 -9426.468} C_VEL
LIN {X 0,Y 434.18,Z 562.77,A -85,B 0,C 180,E1 -9429.591,E2 -9429.591} C_VEL
LIN {X 0,Y 433.659,Z 573.091,A -85,B 0,C 180,E1 -9431.546,E2 -9431.546} C_VEL
LIN {X 0,Y 437.317,Z 596.308,A -85,B 0,C 180,E1 -9432.126,E2 -9432.126} C_VEL
LIN {X 0,Y 436.476,Z 681.147,A -85,B 0,C 180,E1 -9433.544,E2 -9433.544} C_VEL
LIN {X 0,Y 436.005,Z 694.388,A -85,B 0,C 180,E1 -9433.947,E2 -9433.947} C_VEL
LIN {X 0,Y 435.492,Z 706.543,A -85,B 0,C 180,E1 -9434.498,E2 -9434.498} C_VEL
LIN {X 0,Y 434.777,Z 718.815,A -85,B 0,C 180,E1 -9435.252,E2 -9435.252} C_VEL
LIN {X 0,Y 434.103,Z 729.886,A -85,B 0,C 180,E1 -9436.137,E2 -9436.137} C_VEL
LIN {X 0,Y 433.481,Z 740.852,A -85,B 0,C 180,E1 -9437.239,E2 -9437.239} C_VEL
LIN {X 0,Y 432.896,Z 749.391,A -85,B 0,C 180,E1 -9438.292,E2 -9438.292} C_VEL
LIN {X 0,Y 432.35,Z 757.269,A -85,B 0,C 180,E1 -9439.464,E2 -9439.464} C_VEL
LIN {X 0,Y 431.878,Z 764.966,A -85,B 0,C 180,E1 -9440.872,E2 -9440.872} C_VEL
LIN {X 0,Y 431.535,Z 772.063,A -85,B 0,C 180,E1 -9442.515,E2 -9442.515} C_VEL
LIN {X 0,Y 431.293,Z 777.052,A -85,B 0,C 180,E1 -9444.008,E2 -9444.008} C_VEL
LIN {X 0,Y 431.276,Z 780.399,A -85,B 0,C 180,E1 -9445.327,E2 -9445.327} C_VEL
LIN {X 0,Y 431.189,Z 782.26,A -85,B 0,C 180,E1 -9446.263,E2 -9446.263} C_VEL
LIN {X 0,Y 431.236,Z 783.658,A -85,B 0,C 180,E1 -9447.198,E2 -9447.198} C_VEL
LIN {X 0,Y 431.202,Z 784.652,A -85,B 0,C 180,E1 -9448.133,E2 -9448.133} C_VEL
LIN {X 0,Y 431.167,Z 785.473,A -85,B 0,C 180,E1 -9450.001,E2 -9450.001} C_VEL
LIN {X 0,Y 431.203,Z 784.647,A -85,B 0,C 180,E1 -9451.869,E2 -9451.869} C_VEL
LIN {X 0,Y 431.236,Z 783.65,A -85,B 0,C 180,E1 -9452.803,E2 -9452.803} C_VEL
LIN {X 0,Y 431.19,Z 782.25,A -85,B 0,C 180,E1 -9453.739,E2 -9453.739} C_VEL
LIN {X 0,Y 431.304,Z 779.316,A -85,B 0,C 180,E1 -9455.143,E2 -9455.143} C_VEL
LIN {X 0,Y 431.378,Z 775.341,A -85,B 0,C 180,E1 -9456.549,E2 -9456.549} C_VEL
LIN {X 0,Y 431.681,Z 769.226,A -85,B 0,C 180,E1 -9458.191,E2 -9458.191} C_VEL
LIN {X 0,Y 432.013,Z 762.545,A -85,B 0,C 180,E1 -9459.6,E2 -9459.6} C_VEL
LIN {X 0,Y 432.527,Z 754.259,A -85,B 0,C 180,E1 -9461.007,E2 -9461.007} C_VEL
LIN {X 0,Y 433.142,Z 745.768,A -85,B 0,C 180,E1 -9462.178,E2 -9462.178} C_VEL
LIN {X 0,Y 433.714,Z 736.06,A -85,B 0,C 180,E1 -9463.272,E2 -9463.272} C_VEL
LIN {X 0,Y 434.387,Z 724.891,A -85,B 0,C 180,E1 -9464.285,E2 -9464.285} C_VEL
LIN {X 0,Y 435.067,Z 713.518,A -85,B 0,C 180,E1 -9465.099,E2 -9465.099} C_VEL
LIN {X 0,Y 435.704,Z 701.849,A -85,B 0,C 180,E1 -9465.736,E2 -9465.736} C_VEL
LIN {X 0,Y 436.197,Z 689.302,A -85,B 0,C 180,E1 -9466.228,E2 -9466.228} C_VEL
LIN {X 0,Y 436.57,Z 676.578,A -85,B 0,C 180,E1 -9466.544,E2 -9466.544} C_VEL
LIN {X 0,Y 437.286,Z 596.233,A -85,B 0,C 180,E1 -9467.872,E2 -9467.872} C_VEL
LIN {X 0,Y 433.664,Z 573.263,A -85,B 0,C 180,E1 -9468.435,E2 -9468.435} C_VEL
LIN {X 0,Y 433.834,Z 569.222,A -85,B 0,C 180,E1 -9469.151,E2 -9469.151} C_VEL
LIN {X 0,Y 435.037,Z 549.664,A -85,B 0,C 180,E1 -9472.952,E2 -9472.952} C_VEL
LIN {X 0,Y 435.189,Z 545.303,A -85,B 0,C 180,E1 -9473.812,E2 -9473.812} C_VEL
LIN {X 0,Y 433.356,Z 535.129,A -85,B 0,C 180,E1 -9475.969,E2 -9475.969} C_VEL
LIN {X 0,Y 432.457,Z 530.662,A -85,B 0,C 180,E1 -9477.004,E2 -9477.004} C_VEL
LIN {X 0,Y 432.351,Z 530.626,A -85,B 0,C 180,E1 -9480.511,E2 -9480.511} C_VEL
LIN {X 0,Y 432.363,Z 530.629,A -85,B 0,C 180,E1 -9484.004,E2 -9484.004} C_VEL
LIN {X 0,Y 432.326,Z 530.629,A -85,B 0,C 180,E1 -9487.197,E2 -9487.197} C_VEL
LIN {X 0,Y 432.337,Z 530.632,A -85,B 0,C 180,E1 -9490.18,E2 -9490.18} C_VEL
LIN {X 0,Y 432.321,Z 530.632,A -85,B 0,C 180,E1 -9493.061,E2 -9493.061} C_VEL
LIN {X 0,Y 432.337,Z 530.633,A -85,B 0,C 180,E1 -9495.665,E2 -9495.665} C_VEL
LIN {X 0,Y 432.337,Z 530.633,A -85,B 0,C 180,E1 -9498.398,E2 -9498.398} C_VEL
LIN {X 0,Y 432.349,Z 530.632,A -85,B 0,C 180,E1 -9501.851,E2 -9501.851} C_VEL
LIN {X 0,Y 432.345,Z 530.631,A -85,B 0,C 180,E1 -9505.323,E2 -9505.323} C_VEL
LIN {X 0,Y 432.325,Z 530.634,A -85,B 0,C 180,E1 -9508.654,E2 -9508.654} C_VEL
LIN {X 0,Y 432.424,Z 530.824,A -85,B 0,C 180,E1 -9511.015,E2 -9511.015} C_VEL
LIN {X 0,Y 435.171,Z 542.077,A -85,B 0,C 180,E1 -9512.965,E2 -9512.965} C_VEL
LIN {X 0,Y 436.086,Z 548.147,A -85,B 0,C 180,E1 -9513.949,E2 -9513.949} C_VEL
LIN {X 0,Y 435.403,Z 566.38,A -85,B 0,C 180,E1 -9516.677,E2 -9516.677} C_VEL
LIN {X 0,Y 434.603,Z 587.602,A -85,B 0,C 180,E1 -9519.882,E2 -9519.882} C_VEL
LIN {X 0,Y 433.795,Z 611.709,A -85,B 0,C 180,E1 -9523.53,E2 -9523.53} C_VEL
LIN {X 0,Y 433.141,Z 631.496,A -85,B 0,C 180,E1 -9526.512,E2 -9526.512} C_VEL
LIN {X 0,Y 434.725,Z 645.004,A -85,B 0,C 180,E1 -9526.886,E2 -9526.886} C_VEL
LIN {X 0,Y 433.911,Z 704.049,A -85,B 0,C 180,E1 -9528.082,E2 -9528.082} C_VEL
LIN {X 0,Y 433.668,Z 713.994,A -85,B 0,C 180,E1 -9528.431,E2 -9528.431} C_VEL
LIN {X 0,Y 433.393,Z 723.328,A -85,B 0,C 180,E1 -9528.897,E2 -9528.897} C_VEL
LIN {X 0,Y 433.023,Z 733.544,A -85,B 0,C 180,E1 -9529.598,E2 -9529.598} C_VEL
LIN {X 0,Y 432.7,Z 741.441,A -85,B 0,C 180,E1 -9530.299,E2 -9530.299} C_VEL
LIN {X 0,Y 432.342,Z 748.933,A -85,B 0,C 180,E1 -9531.116,E2 -9531.116} C_VEL
LIN {X 0,Y 431.948,Z 757.423,A -85,B 0,C 180,E1 -9532.286,E2 -9532.286} C_VEL
LIN {X 0,Y 431.701,Z 763.909,A -85,B 0,C 180,E1 -9533.456,E2 -9533.456} C_VEL
LIN {X 0,Y 431.588,Z 768.083,A -85,B 0,C 180,E1 -9534.393,E2 -9534.393} C_VEL
LIN {X 0,Y 431.36,Z 771.461,A -85,B 0,C 180,E1 -9535.327,E2 -9535.327} C_VEL
LIN {X 0,Y 431.317,Z 774.126,A -85,B 0,C 180,E1 -9536.263,E2 -9536.263} C_VEL
LIN {X 0,Y 431.305,Z 776.145,A -85,B 0,C 180,E1 -9537.198,E2 -9537.198} C_VEL
LIN {X 0,Y 431.206,Z 777.567,A -85,B 0,C 180,E1 -9538.132,E2 -9538.132} C_VEL
LIN {X 0,Y 431.147,Z 778.416,A -85,B 0,C 180,E1 -9539.066,E2 -9539.066} C_VEL
LIN {X 0,Y 431.143,Z 778.69,A -85,B 0,C 180,E1 -9540,E2 -9540} C_VEL
LIN {X 0,Y 431.148,Z 778.365,A -85,B 0,C 180,E1 -9540.934,E2 -9540.934} C_VEL
LIN {X 0,Y 431.205,Z 777.446,A -85,B 0,C 180,E1 -9541.868,E2 -9541.868} C_VEL
LIN {X 0,Y 431.324,Z 774.999,A -85,B 0,C 180,E1 -9543.269,E2 -9543.269} C_VEL
LIN {X 0,Y 431.345,Z 771.082,A -85,B 0,C 180,E1 -9544.673,E2 -9544.673} C_VEL
LIN {X 0,Y 431.494,Z 767.606,A -85,B 0,C 180,E1 -9545.608,E2 -9545.608} C_VEL
LIN {X 0,Y 431.624,Z 762.743,A -85,B 0,C 180,E1 -9546.661,E2 -9546.661} C_VEL
LIN {X 0,Y 431.864,Z 756.666,A -85,B 0,C 180,E1 -9547.716,E2 -9547.716} C_VEL
LIN {X 0,Y 432.121,Z 749.86,A -85,B 0,C 180,E1 -9548.653,E2 -9548.653} C_VEL
LIN {X 0,Y 432.469,Z 742.54,A -85,B 0,C 180,E1 -9549.471,E2 -9549.471} C_VEL
LIN {X 0,Y 432.751,Z 734.844,A -85,B 0,C 180,E1 -9550.173,E2 -9550.173} C_VEL
LIN {X 0,Y 433.134,Z 724.203,A -85,B 0,C 180,E1 -9550.932,E2 -9550.932} C_VEL
LIN {X 0,Y 433.391,Z 713.705,A -85,B 0,C 180,E1 -9551.458,E2 -9551.458} C_VEL
LIN {X 0,Y 433.632,Z 703.577,A -85,B 0,C 180,E1 -9551.807,E2 -9551.807} C_VEL
LIN {X 0,Y 434.214,Z 644.067,A -85,B 0,C 180,E1 -9552.958,E2 -9552.958} C_VEL
LIN {X 0,Y 432.822,Z 631.419,A -85,B 0,C 180,E1 -9553.266,E2 -9553.266} C_VEL
LIN {X 0,Y 433.519,Z 610.345,A -85,B 0,C 180,E1 -9556.481,E2 -9556.481} C_VEL
LIN {X 0,Y 434.334,Z 587.098,A -85,B 0,C 180,E1 -9560.067,E2 -9560.067} C_VEL
LIN {X 0,Y 435.238,Z 564.545,A -85,B 0,C 180,E1 -9563.556,E2 -9563.556} C_VEL
LIN {X 0,Y 435.875,Z 548.375,A -85,B 0,C 180,E1 -9566.064,E2 -9566.064} C_VEL
LIN {X 0,Y 434.269,Z 539.466,A -85,B 0,C 180,E1 -9567.541,E2 -9567.541} C_VEL
LIN {X 0,Y 432.418,Z 530.731,A -85,B 0,C 180,E1 -9569.053,E2 -9569.053} C_VEL
LIN {X 0,Y 432.327,Z 530.635,A -85,B 0,C 180,E1 -9572.443,E2 -9572.443} C_VEL
LIN {X 0,Y 432.35,Z 530.627,A -85,B 0,C 180,E1 -9575.632,E2 -9575.632} C_VEL
LIN {X 0,Y 432.351,Z 530.629,A -85,B 0,C 180,E1 -9578.715,E2 -9578.715} C_VEL
LIN {X 0,Y 432.338,Z 530.614,A -85,B 0,C 180,E1 -9581.797,E2 -9581.797} C_VEL
LIN {X 0,Y 432.338,Z 530.614,A -85,B 0,C 180,E1 -9584.347,E2 -9584.347} C_VEL
LIN {X 0,Y 432.33,Z 530.631,A -85,B 0,C 180,E1 -9587.015,E2 -9587.015} C_VEL
LIN {X 0,Y 432.338,Z 530.617,A -85,B 0,C 180,E1 -9589.82,E2 -9589.82} C_VEL
LIN {X 0,Y 432.311,Z 530.635,A -85,B 0,C 180,E1 -9593.022,E2 -9593.022} C_VEL
LIN {X 0,Y 432.364,Z 530.62,A -85,B 0,C 180,E1 -9595.996,E2 -9595.996} C_VEL
LIN {X 0,Y 432.352,Z 530.628,A -85,B 0,C 180,E1 -9599.489,E2 -9599.489} C_VEL
LIN {X 0,Y 432.395,Z 530.624,A -85,B 0,C 180,E1 -9602.928,E2 -9602.928} C_VEL
LIN {X 0,Y 432.374,Z 530.622,A -85,B 0,C 180,E1 -9606.531,E2 -9606.531} C_VEL
LIN {X 0,Y 432.402,Z 530.883,A -85,B 0,C 180,E1 -9607.04,E2 -9607.04} C_VEL
LIN {X 0,Y 434.043,Z 539.212,A -85,B 0,C 180,E1 -9609.131,E2 -9609.131} C_VEL
LIN {X 0,Y 434.152,Z 543.45,A -85,B 0,C 180,E1 -9610.126,E2 -9610.126} C_VEL
LIN {X 0,Y 433.806,Z 550.172,A -85,B 0,C 180,E1 -9611.608,E2 -9611.608} C_VEL
LIN {X 0,Y 435.262,Z 557.33,A -85,B 0,C 180,E1 -9611.832,E2 -9611.832} C_VEL
LIN {X 0,Y 437.556,Z 569.554,A -85,B 0,C 180,E1 -9612.139,E2 -9612.139} C_VEL
LIN {X 0,Y 437.216,Z 604.316,A -85,B 0,C 180,E1 -9612.712,E2 -9612.712} C_VEL
LIN {X 0,Y 436.448,Z 610.156,A -85,B 0,C 180,E1 -9612.779,E2 -9612.779} C_VEL
LIN {X 0,Y 430.867,Z 629.159,A -85,B 0,C 180,E1 -9612.871,E2 -9612.871} C_VEL
LIN {X 0,Y 430.16,Z 634.997,A -85,B 0,C 180,E1 -9612.941,E2 -9612.941} C_VEL
LIN {X 0,Y 429.742,Z 658.744,A -85,B 0,C 180,E1 -9613.369,E2 -9613.369} C_VEL
LIN {X 0,Y 429.348,Z 672.218,A -85,B 0,C 180,E1 -9613.812,E2 -9613.812} C_VEL
LIN {X 0,Y 428.812,Z 684.85,A -85,B 0,C 180,E1 -9614.432,E2 -9614.432} C_VEL
LIN {X 0,Y 428.118,Z 697.262,A -85,B 0,C 180,E1 -9615.258,E2 -9615.258} C_VEL
LIN {X 0,Y 427.552,Z 708.072,A -85,B 0,C 180,E1 -9616.186,E2 -9616.186} C_VEL
LIN {X 0,Y 426.914,Z 717.284,A -85,B 0,C 180,E1 -9617.159,E2 -9617.159} C_VEL
LIN {X 0,Y 426.206,Z 726.469,A -85,B 0,C 180,E1 -9618.345,E2 -9618.345} C_VEL
LIN {X 0,Y 425.569,Z 735.384,A -85,B 0,C 180,E1 -9619.773,E2 -9619.773} C_VEL
LIN {X 0,Y 425.066,Z 742.56,A -85,B 0,C 180,E1 -9621.202,E2 -9621.202} C_VEL
LIN {X 0,Y 424.684,Z 747.404,A -85,B 0,C 180,E1 -9622.391,E2 -9622.391} C_VEL
LIN {X 0,Y 424.572,Z 751.51,A -85,B 0,C 180,E1 -9623.622,E2 -9623.622} C_VEL
LIN {X 0,Y 424.285,Z 755.702,A -85,B 0,C 180,E1 -9625.248,E2 -9625.248} C_VEL
LIN {X 0,Y 424.239,Z 757.56,A -85,B 0,C 180,E1 -9626.2,E2 -9626.2} C_VEL
LIN {X 0,Y 424.241,Z 758.96,A -85,B 0,C 180,E1 -9627.15,E2 -9627.15} C_VEL
LIN {X 0,Y 424.092,Z 760.576,A -85,B 0,C 180,E1 -9629.05,E2 -9629.05} C_VEL
LIN {X 0,Y 424.085,Z 760.811,A -85,B 0,C 180,E1 -9629.999,E2 -9629.999} C_VEL
LIN {X 0,Y 424.091,Z 760.624,A -85,B 0,C 180,E1 -9630.949,E2 -9630.949} C_VEL
LIN {X 0,Y 424.237,Z 759.075,A -85,B 0,C 180,E1 -9632.848,E2 -9632.848} C_VEL
LIN {X 0,Y 424.225,Z 757.723,A -85,B 0,C 180,E1 -9633.799,E2 -9633.799} C_VEL
LIN {X 0,Y 424.373,Z 754.856,A -85,B 0,C 180,E1 -9635.225,E2 -9635.225} C_VEL
LIN {X 0,Y 424.583,Z 750.827,A -85,B 0,C 180,E1 -9636.701,E2 -9636.701} C_VEL
LIN {X 0,Y 424.818,Z 745.962,A -85,B 0,C 180,E1 -9638.083,E2 -9638.083} C_VEL
LIN {X 0,Y 425.313,Z 739.652,A -85,B 0,C 180,E1 -9639.51,E2 -9639.51} C_VEL
LIN {X 0,Y 425.874,Z 731.752,A -85,B 0,C 180,E1 -9640.939,E2 -9640.939} C_VEL
LIN {X 0,Y 426.385,Z 723.702,A -85,B 0,C 180,E1 -9642.13,E2 -9642.13} C_VEL
LIN {X 0,Y 427.181,Z 713.868,A -85,B 0,C 180,E1 -9643.315,E2 -9643.315} C_VEL
LIN {X 0,Y 427.8,Z 702.821,A -85,B 0,C 180,E1 -9644.386,E2 -9644.386} C_VEL
LIN {X 0,Y 428.467,Z 691.979,A -85,B 0,C 180,E1 -9645.214,E2 -9645.214} C_VEL
LIN {X 0,Y 429.08,Z 679.996,A -85,B 0,C 180,E1 -9645.922,E2 -9645.922} C_VEL
LIN {X 0,Y 429.537,Z 667.732,A -85,B 0,C 180,E1 -9646.454,E2 -9646.454} C_VEL
LIN {X 0,Y 429.891,Z 655.129,A -85,B 0,C 180,E1 -9646.807,E2 -9646.807} C_VEL
LIN {X 0,Y 430.672,Z 569.279,A -85,B 0,C 180,E1 -9648.26,E2 -9648.26} C_VEL
LIN {X 0,Y 426.954,Z 550.775,A -85,B 0,C 180,E1 -9648.768,E2 -9648.768} C_VEL
LIN {X 0,Y 426.935,Z 549.274,A -85,B 0,C 180,E1 -9648.995,E2 -9648.995} C_VEL
LIN {X 0,Y 427.227,Z 542.145,A -85,B 0,C 180,E1 -9650.661,E2 -9650.661} C_VEL
LIN {X 0,Y 425.548,Z 532.513,A -85,B 0,C 180,E1 -9653.08,E2 -9653.08} C_VEL
LIN {X 0,Y 425.349,Z 531.52,A -85,B 0,C 180,E1 -9653.426,E2 -9653.426} C_VEL
LIN {X 0,Y 425.347,Z 531.498,A -85,B 0,C 180,E1 -9656.843,E2 -9656.843} C_VEL
LIN {X 0,Y 425.29,Z 531.499,A -85,B 0,C 180,E1 -9659.718,E2 -9659.718} C_VEL
LIN {X 0,Y 425.28,Z 531.508,A -85,B 0,C 180,E1 -9663.047,E2 -9663.047} C_VEL
LIN {X 0,Y 425.282,Z 531.505,A -85,B 0,C 180,E1 -9665.928,E2 -9665.928} C_VEL
LIN {X 0,Y 425.301,Z 531.507,A -85,B 0,C 180,E1 -9669.043,E2 -9669.043} C_VEL
LIN {X 0,Y 425.288,Z 531.508,A -85,B 0,C 180,E1 -9671.958,E2 -9671.958} C_VEL
LIN {X 0,Y 425.282,Z 531.5,A -85,B 0,C 180,E1 -9675.282,E2 -9675.282} C_VEL
LIN {X 0,Y 425.3,Z 531.505,A -85,B 0,C 180,E1 -9678.624,E2 -9678.624} C_VEL
LIN {X 0,Y 425.319,Z 531.492,A -85,B 0,C 180,E1 -9681.103,E2 -9681.103} C_VEL
LIN {X 0,Y 425.298,Z 531.505,A -85,B 0,C 180,E1 -9684.664,E2 -9684.664} C_VEL
LIN {X 0,Y 425.26,Z 531.509,A -85,B 0,C 180,E1 -9688.072,E2 -9688.072} C_VEL
LIN {X 0,Y 425.331,Z 531.503,A -85,B 0,C 180,E1 -9691.368,E2 -9691.368} C_VEL
LIN {X 0,Y 425.289,Z 531.505,A -85,B 0,C 180,E1 -9694.554,E2 -9694.554} C_VEL
LIN {X 0,Y 425.281,Z 531.505,A -85,B 0,C 180,E1 -9697.661,E2 -9697.661} C_VEL
LIN {X 0,Y 425.355,Z 531.497,A -85,B 0,C 180,E1 -9700.704,E2 -9700.704} C_VEL
LIN {X 0,Y 425.381,Z 531.491,A -85,B 0,C 180,E1 -9703.688,E2 -9703.688} C_VEL
LIN {X 0,Y 425.404,Z 531.495,A -85,B 0,C 180,E1 -9707.598,E2 -9707.598} C_VEL
LIN {X 0,Y 425.435,Z 531.486,A -85,B 0,C 180,E1 -9711.45,E2 -9711.45} C_VEL
LIN {X 0,Y 425.547,Z 531.473,A -85,B 0,C 180,E1 -9714.313,E2 -9714.313} C_VEL
LIN {X 0,Y 425.568,Z 531.47,A -85,B 0,C 180,E1 -9718.107,E2 -9718.107} C_VEL
LIN {X 0,Y 425.697,Z 531.457,A -85,B 0,C 180,E1 -9720,E2 -9720} C_VEL
LIN {X 0,Y 425.55,Z 531.469,A -85,B 0,C 180,E1 -9722.84,E2 -9722.84} C_VEL
LIN {X 0,Y 425.566,Z 531.476,A -85,B 0,C 180,E1 -9725.687,E2 -9725.687} C_VEL
LIN {X 0,Y 425.435,Z 531.485,A -85,B 0,C 180,E1 -9728.55,E2 -9728.55} C_VEL
LIN {X 0,Y 425.422,Z 531.488,A -85,B 0,C 180,E1 -9732.402,E2 -9732.402} C_VEL
LIN {X 0,Y 425.381,Z 531.489,A -85,B 0,C 180,E1 -9736.312,E2 -9736.312} C_VEL
LIN {X 0,Y 425.353,Z 531.503,A -85,B 0,C 180,E1 -9739.648,E2 -9739.648} C_VEL
LIN {X 0,Y 425.3,Z 531.506,A -85,B 0,C 180,E1 -9743.366,E2 -9743.366} C_VEL
LIN {X 0,Y 425.342,Z 531.494,A -85,B 0,C 180,E1 -9746.845,E2 -9746.845} C_VEL
LIN {X 0,Y 425.284,Z 531.51,A -85,B 0,C 180,E1 -9749.72,E2 -9749.72} C_VEL
LIN {X 0,Y 425.278,Z 531.508,A -85,B 0,C 180,E1 -9753.048,E2 -9753.048} C_VEL
LIN {X 0,Y 425.279,Z 531.496,A -85,B 0,C 180,E1 -9755.93,E2 -9755.93} C_VEL
LIN {X 0,Y 425.298,Z 531.505,A -85,B 0,C 180,E1 -9759.045,E2 -9759.045} C_VEL
LIN {X 0,Y 425.269,Z 531.499,A -85,B 0,C 180,E1 -9762.654,E2 -9762.654} C_VEL
LIN {X 0,Y 425.314,Z 531.501,A -85,B 0,C 180,E1 -9766.053,E2 -9766.053} C_VEL
LIN {X 0,Y 425.306,Z 531.505,A -85,B 0,C 180,E1 -9768.627,E2 -9768.627} C_VEL
LIN {X 0,Y 425.32,Z 531.495,A -85,B 0,C 180,E1 -9771.105,E2 -9771.105} C_VEL
LIN {X 0,Y 425.297,Z 531.507,A -85,B 0,C 180,E1 -9774.665,E2 -9774.665} C_VEL
LIN {X 0,Y 425.262,Z 531.465,A -85,B 0,C 180,E1 -9778.074,E2 -9778.074} C_VEL
LIN {X 0,Y 425.33,Z 531.504,A -85,B 0,C 180,E1 -9781.369,E2 -9781.369} C_VEL
LIN {X 0,Y 425.366,Z 531.545,A -85,B 0,C 180,E1 -9782.734,E2 -9782.734} C_VEL
LIN {X 0,Y 427.366,Z 541.365,A -85,B 0,C 180,E1 -9784.953,E2 -9784.953} C_VEL
LIN {X 0,Y 428.284,Z 547.687,A -85,B 0,C 180,E1 -9786.296,E2 -9786.296} C_VEL
LIN {X 0,Y 427.271,Z 562.799,A -85,B 0,C 180,E1 -9789.291,E2 -9789.291} C_VEL
LIN {X 0,Y 426.71,Z 572.905,A -85,B 0,C 180,E1 -9791.236,E2 -9791.236} C_VEL
LIN {X 0,Y 430.548,Z 596.993,A -85,B 0,C 180,E1 -9791.851,E2 -9791.851} C_VEL
LIN {X 0,Y 429.674,Z 680.954,A -85,B 0,C 180,E1 -9793.276,E2 -9793.276} C_VEL
LIN {X 0,Y 429.19,Z 694.191,A -85,B 0,C 180,E1 -9793.685,E2 -9793.685} C_VEL
LIN {X 0,Y 428.629,Z 706.343,A -85,B 0,C 180,E1 -9794.244,E2 -9794.244} C_VEL
LIN {X 0,Y 427.918,Z 718.615,A -85,B 0,C 180,E1 -9795.01,E2 -9795.01} C_VEL
LIN {X 0,Y 427.179,Z 729.554,A -85,B 0,C 180,E1 -9795.896,E2 -9795.896} C_VEL
LIN {X 0,Y 426.503,Z 740.648,A -85,B 0,C 180,E1 -9797.027,E2 -9797.027} C_VEL
LIN {X 0,Y 425.907,Z 749.188,A -85,B 0,C 180,E1 -9798.097,E2 -9798.097} C_VEL
LIN {X 0,Y 425.319,Z 757.064,A -85,B 0,C 180,E1 -9799.288,E2 -9799.288} C_VEL
LIN {X 0,Y 424.834,Z 764.762,A -85,B 0,C 180,E1 -9800.719,E2 -9800.719} C_VEL
LIN {X 0,Y 424.452,Z 771.858,A -85,B 0,C 180,E1 -9802.389,E2 -9802.389} C_VEL
LIN {X 0,Y 424.247,Z 776.207,A -85,B 0,C 180,E1 -9803.695,E2 -9803.695} C_VEL
LIN {X 0,Y 424.205,Z 780.195,A -85,B 0,C 180,E1 -9805.249,E2 -9805.249} C_VEL
LIN {X 0,Y 424.101,Z 782.056,A -85,B 0,C 180,E1 -9806.2,E2 -9806.2} C_VEL
LIN {X 0,Y 424.132,Z 783.453,A -85,B 0,C 180,E1 -9807.151,E2 -9807.151} C_VEL
LIN {X 0,Y 424.128,Z 784.448,A -85,B 0,C 180,E1 -9808.102,E2 -9808.102} C_VEL
LIN {X 0,Y 424.084,Z 785.269,A -85,B 0,C 180,E1 -9810.001,E2 -9810.001} C_VEL
LIN {X 0,Y 424.088,Z 785.064,A -85,B 0,C 180,E1 -9810.95,E2 -9810.95} C_VEL
LIN {X 0,Y 424.129,Z 784.443,A -85,B 0,C 180,E1 -9811.9,E2 -9811.9} C_VEL
LIN {X 0,Y 424.132,Z 783.445,A -85,B 0,C 180,E1 -9812.85,E2 -9812.85} C_VEL
LIN {X 0,Y 424.101,Z 782.045,A -85,B 0,C 180,E1 -9813.802,E2 -9813.802} C_VEL
LIN {X 0,Y 424.217,Z 779.11,A -85,B 0,C 180,E1 -9815.229,E2 -9815.229} C_VEL
LIN {X 0,Y 424.303,Z 775.135,A -85,B 0,C 180,E1 -9816.659,E2 -9816.659} C_VEL
LIN {X 0,Y 424.615,Z 769.019,A -85,B 0,C 180,E1 -9818.328,E2 -9818.328} C_VEL
LIN {X 0,Y 424.968,Z 762.338,A -85,B 0,C 180,E1 -9819.76,E2 -9819.76} C_VEL
LIN {X 0,Y 425.51,Z 754.051,A -85,B 0,C 180,E1 -9821.191,E2 -9821.191} C_VEL
LIN {X 0,Y 426.171,Z 745.56,A -85,B 0,C 180,E1 -9822.38,E2 -9822.38} C_VEL
LIN {X 0,Y 426.84,Z 735.146,A -85,B 0,C 180,E1 -9823.562,E2 -9823.562} C_VEL
LIN {X 0,Y 427.482,Z 724.682,A -85,B 0,C 180,E1 -9824.521,E2 -9824.521} C_VEL
LIN {X 0,Y 428.211,Z 713.309,A -85,B 0,C 180,E1 -9825.347,E2 -9825.347} C_VEL
LIN {X 0,Y 428.881,Z 701.638,A -85,B 0,C 180,E1 -9825.993,E2 -9825.993} C_VEL
LIN {X 0,Y 429.397,Z 689.089,A -85,B 0,C 180,E1 -9826.492,E2 -9826.492} C_VEL
LIN {X 0,Y 429.769,Z 676.358,A -85,B 0,C 180,E1 -9826.813,E2 -9826.813} C_VEL
LIN {X 0,Y 430.412,Z 596.329,A -85,B 0,C 180,E1 -9828.162,E2 -9828.162} C_VEL
LIN {X 0,Y 426.736,Z 573.068,A -85,B 0,C 180,E1 -9828.744,E2 -9828.744} C_VEL
LIN {X 0,Y 426.93,Z 569.018,A -85,B 0,C 180,E1 -9829.473,E2 -9829.473} C_VEL
LIN {X 0,Y 428.134,Z 550.172,A -85,B 0,C 180,E1 -9833.202,E2 -9833.202} C_VEL
LIN {X 0,Y 428.238,Z 546.381,A -85,B 0,C 180,E1 -9833.966,E2 -9833.966} C_VEL
LIN {X 0,Y 426.076,Z 534.941,A -85,B 0,C 180,E1 -9836.447,E2 -9836.447} C_VEL
LIN {X 0,Y 425.376,Z 531.54,A -85,B 0,C 180,E1 -9837.268,E2 -9837.268} C_VEL
LIN {X 0,Y 425.294,Z 531.51,A -85,B 0,C 180,E1 -9840.762,E2 -9840.762} C_VEL
LIN {X 0,Y 425.315,Z 531.509,A -85,B 0,C 180,E1 -9844.288,E2 -9844.288} C_VEL
LIN {X 0,Y 425.283,Z 531.509,A -85,B 0,C 180,E1 -9847.695,E2 -9847.695} C_VEL
LIN {X 0,Y 425.283,Z 531.508,A -85,B 0,C 180,E1 -9850.521,E2 -9850.521} C_VEL
LIN {X 0,Y 425.262,Z 531.512,A -85,B 0,C 180,E1 -9853.351,E2 -9853.351} C_VEL
LIN {X 0,Y 425.262,Z 531.513,A -85,B 0,C 180,E1 -9856.649,E2 -9856.649} C_VEL
LIN {X 0,Y 425.291,Z 531.51,A -85,B 0,C 180,E1 -9859.873,E2 -9859.873} C_VEL
LIN {X 0,Y 425.288,Z 531.51,A -85,B 0,C 180,E1 -9862.488,E2 -9862.488} C_VEL
LIN {X 0,Y 425.312,Z 531.508,A -85,B 0,C 180,E1 -9865.818,E2 -9865.818} C_VEL
LIN {X 0,Y 425.294,Z 531.512,A -85,B 0,C 180,E1 -9869.239,E2 -9869.239} C_VEL
LIN {X 0,Y 425.344,Z 531.718,A -85,B 0,C 180,E1 -9870.594,E2 -9870.594} C_VEL
LIN {X 0,Y 428.063,Z 542.053,A -85,B 0,C 180,E1 -9872.447,E2 -9872.447} C_VEL
LIN {X 0,Y 429.354,Z 549.99,A -85,B 0,C 180,E1 -9873.771,E2 -9873.771} C_VEL
LIN {X 0,Y 428.623,Z 567.94,A -85,B 0,C 180,E1 -9876.5,E2 -9876.5} C_VEL
LIN {X 0,Y 427.673,Z 591.223,A -85,B 0,C 180,E1 -9880.063,E2 -9880.063} C_VEL
LIN {X 0,Y 426.746,Z 616.862,A -85,B 0,C 180,E1 -9883.987,E2 -9883.987} C_VEL
LIN {X 0,Y 426.233,Z 631.71,A -85,B 0,C 180,E1 -9886.236,E2 -9886.236} C_VEL
LIN {X 0,Y 427.934,Z 646.166,A -85,B 0,C 180,E1 -9886.641,E2 -9886.641} C_VEL
LIN {X 0,Y 427.044,Z 704.294,A -85,B 0,C 180,E1 -9887.857,E2 -9887.857} C_VEL
LIN {X 0,Y 426.773,Z 713.42,A -85,B 0,C 180,E1 -9888.181,E2 -9888.181} C_VEL
LIN {X 0,Y 426.456,Z 723.899,A -85,B 0,C 180,E1 -9888.714,E2 -9888.714} C_VEL
LIN {X 0,Y 426.069,Z 733.902,A -85,B 0,C 180,E1 -9889.426,E2 -9889.426} C_VEL
LIN {X 0,Y 425.684,Z 742.906,A -85,B 0,C 180,E1 -9890.257,E2 -9890.257} C_VEL
LIN {X 0,Y 425.222,Z 751.139,A -85,B 0,C 180,E1 -9891.206,E2 -9891.206} C_VEL
LIN {X 0,Y 424.934,Z 757.633,A -85,B 0,C 180,E1 -9892.158,E2 -9892.158} C_VEL
LIN {X 0,Y 424.651,Z 764.11,A -85,B 0,C 180,E1 -9893.347,E2 -9893.347} C_VEL
LIN {X 0,Y 424.541,Z 768.265,A -85,B 0,C 180,E1 -9894.3,E2 -9894.3} C_VEL
LIN {X 0,Y 424.296,Z 771.624,A -85,B 0,C 180,E1 -9895.249,E2 -9895.249} C_VEL
LIN {X 0,Y 424.225,Z 774.268,A -85,B 0,C 180,E1 -9896.2,E2 -9896.2} C_VEL
LIN {X 0,Y 424.211,Z 776.267,A -85,B 0,C 180,E1 -9897.151,E2 -9897.151} C_VEL
LIN {X 0,Y 424.134,Z 777.665,A -85,B 0,C 180,E1 -9898.101,E2 -9898.101} C_VEL
LIN {X 0,Y 424.068,Z 778.487,A -85,B 0,C 180,E1 -9899.05,E2 -9899.05} C_VEL
LIN {X 0,Y 424.061,Z 778.74,A -85,B 0,C 180,E1 -9900,E2 -9900} C_VEL
LIN {X 0,Y 424.069,Z 778.397,A -85,B 0,C 180,E1 -9900.95,E2 -9900.95} C_VEL
LIN {X 0,Y 424.132,Z 777.455,A -85,B 0,C 180,E1 -9901.899,E2 -9901.899} C_VEL
LIN {X 0,Y 424.218,Z 774.939,A -85,B 0,C 180,E1 -9903.324,E2 -9903.324} C_VEL
LIN {X 0,Y 424.28,Z 770.98,A -85,B 0,C 180,E1 -9904.751,E2 -9904.751} C_VEL
LIN {X 0,Y 424.436,Z 766.27,A -85,B 0,C 180,E1 -9905.996,E2 -9905.996} C_VEL
LIN {X 0,Y 424.688,Z 760.627,A -85,B 0,C 180,E1 -9907.13,E2 -9907.13} C_VEL
LIN {X 0,Y 424.861,Z 754.722,A -85,B 0,C 180,E1 -9908.083,E2 -9908.083} C_VEL
LIN {X 0,Y 425.188,Z 747.484,A -85,B 0,C 180,E1 -9909.034,E2 -9909.034} C_VEL
LIN {X 0,Y 425.583,Z 738.457,A -85,B 0,C 180,E1 -9909.985,E2 -9909.985} C_VEL
LIN {X 0,Y 425.954,Z 729.598,A -85,B 0,C 180,E1 -9910.697,E2 -9910.697} C_VEL
LIN {X 0,Y 426.214,Z 720.047,A -85,B 0,C 180,E1 -9911.292,E2 -9911.292} C_VEL
LIN {X 0,Y 426.521,Z 708.765,A -85,B 0,C 180,E1 -9911.796,E2 -9911.796} C_VEL
LIN {X 0,Y 426.642,Z 697.672,A -85,B 0,C 180,E1 -9912.094,E2 -9912.094} C_VEL
LIN {X 0,Y 427.224,Z 644.667,A -85,B 0,C 180,E1 -9913.123,E2 -9913.123} C_VEL
LIN {X 0,Y 425.812,Z 631.434,A -85,B 0,C 180,E1 -9913.451,E2 -9913.451} C_VEL
LIN {X 0,Y 426.596,Z 608.444,A -85,B 0,C 180,E1 -9916.995,E2 -9916.995} C_VEL
LIN {X 0,Y 427.401,Z 586.602,A -85,B 0,C 180,E1 -9920.399,E2 -9920.399} C_VEL
LIN {X 0,Y 428.28,Z 565.43,A -85,B 0,C 180,E1 -9923.706,E2 -9923.706} C_VEL
LIN {X 0,Y 428.902,Z 549.172,A -85,B 0,C 180,E1 -9926.259,E2 -9926.259} C_VEL
LIN {X 0,Y 426.565,Z 537.205,A -85,B 0,C 180,E1 -9928.273,E2 -9928.273} C_VEL
LIN {X 0,Y 425.384,Z 531.615,A -85,B 0,C 180,E1 -9929.266,E2 -9929.266} C_VEL
LIN {X 0,Y 425.287,Z 531.509,A -85,B 0,C 180,E1 -9933.048,E2 -9933.048} C_VEL
LIN {X 0,Y 425.29,Z 531.509,A -85,B 0,C 180,E1 -9935.929,E2 -9935.929} C_VEL
LIN {X 0,Y 425.301,Z 531.504,A -85,B 0,C 180,E1 -9939.043,E2 -9939.043} C_VEL
LIN {X 0,Y 425.279,Z 531.484,A -85,B 0,C 180,E1 -9942.653,E2 -9942.653} C_VEL
LIN {X 0,Y 425.273,Z 531.507,A -85,B 0,C 180,E1 -9946.045,E2 -9946.045} C_VEL
LIN {X 0,Y 425.28,Z 531.503,A -85,B 0,C 180,E1 -9948.621,E2 -9948.621} C_VEL
LIN {X 0,Y 425.306,Z 531.493,A -85,B 0,C 180,E1 -9951.101,E2 -9951.101} C_VEL
LIN {X 0,Y 425.304,Z 531.503,A -85,B 0,C 180,E1 -9954.664,E2 -9954.664} C_VEL
LIN {X 0,Y 425.27,Z 531.511,A -85,B 0,C 180,E1 -9958.073,E2 -9958.073} C_VEL
LIN {X 0,Y 425.336,Z 531.5,A -85,B 0,C 180,E1 -9961.367,E2 -9961.367} C_VEL
LIN {X 0,Y 425.296,Z 531.509,A -85,B 0,C 180,E1 -9964.554,E2 -9964.554} C_VEL
LIN {X 0,Y 425.362,Z 531.64,A -85,B 0,C 180,E1 -9966.764,E2 -9966.764} C_VEL
LIN {X 0,Y 427.195,Z 541.523,A -85,B 0,C 180,E1 -9969.286,E2 -9969.286} C_VEL
LIN {X 0,Y 426.942,Z 549,A -85,B 0,C 180,E1 -9971.037,E2 -9971.037} C_VEL
LIN {X 0,Y 426.901,Z 550.628,A -85,B 0,C 180,E1 -9971.321,E2 -9971.321} C_VEL
LIN {X 0,Y 430.812,Z 570.048,A -85,B 0,C 180,E1 -9971.854,E2 -9971.854} C_VEL
LIN {X 0,Y 430.16,Z 634.997,A -85,B 0,C 180,E1 -9972.941,E2 -9972.941} C_VEL
LIN {X 0,Y 429.424,Z 640.848,A -85,B 0,C 180,E1 -9973.008,E2 -9973.008} C_VEL
LIN {X 0,Y 423.568,Z 659.783,A -85,B 0,C 180,E1 -9973.14,E2 -9973.14} C_VEL
LIN {X 0,Y 422.816,Z 665.53,A -85,B 0,C 180,E1 -9973.289,E2 -9973.289} C_VEL
LIN {X 0,Y 422.337,Z 678.403,A -85,B 0,C 180,E1 -9973.815,E2 -9973.815} C_VEL
LIN {X 0,Y 421.799,Z 689.018,A -85,B 0,C 180,E1 -9974.414,E2 -9974.414} C_VEL
LIN {X 0,Y 421.11,Z 700.486,A -85,B 0,C 180,E1 -9975.255,E2 -9975.255} C_VEL
LIN {X 0,Y 420.444,Z 711.653,A -85,B 0,C 180,E1 -9976.299,E2 -9976.299} C_VEL
LIN {X 0,Y 419.684,Z 721.395,A -85,B 0,C 180,E1 -9977.425,E2 -9977.425} C_VEL
LIN {X 0,Y 419.048,Z 729.894,A -85,B 0,C 180,E1 -9978.634,E2 -9978.634} C_VEL
LIN {X 0,Y 418.407,Z 738.15,A -85,B 0,C 180,E1 -9980.085,E2 -9980.085} C_VEL
LIN {X 0,Y 417.858,Z 744.801,A -85,B 0,C 180,E1 -9981.536,E2 -9981.536} C_VEL
LIN {X 0,Y 417.523,Z 751.033,A -85,B 0,C 180,E1 -9983.279,E2 -9983.279} C_VEL
LIN {X 0,Y 417.326,Z 754.845,A -85,B 0,C 180,E1 -9984.685,E2 -9984.685} C_VEL
LIN {X 0,Y 417.146,Z 757.766,A -85,B 0,C 180,E1 -9986.135,E2 -9986.135} C_VEL
LIN {X 0,Y 417.158,Z 759.165,A -85,B 0,C 180,E1 -9987.102,E2 -9987.102} C_VEL
LIN {X 0,Y 417.014,Z 760.78,A -85,B 0,C 180,E1 -9989.033,E2 -9989.033} C_VEL
LIN {X 0,Y 417.004,Z 761.015,A -85,B 0,C 180,E1 -9989.999,E2 -9989.999} C_VEL
LIN {X 0,Y 417.014,Z 760.828,A -85,B 0,C 180,E1 -9990.965,E2 -9990.965} C_VEL
LIN {X 0,Y 417.154,Z 759.279,A -85,B 0,C 180,E1 -9992.896,E2 -9992.896} C_VEL
LIN {X 0,Y 417.133,Z 757.927,A -85,B 0,C 180,E1 -9993.863,E2 -9993.863} C_VEL
LIN {X 0,Y 417.32,Z 755.059,A -85,B 0,C 180,E1 -9995.314,E2 -9995.314} C_VEL
LIN {X 0,Y 417.52,Z 751.173,A -85,B 0,C 180,E1 -9996.766,E2 -9996.766} C_VEL
LIN {X 0,Y 417.788,Z 746.165,A -85,B 0,C 180,E1 -9998.22,E2 -9998.22} C_VEL
LIN {X 0,Y 418.31,Z 739.855,A -85,B 0,C 180,E1 -9999.671,E2 -9999.671} C_VEL
LIN {X 0,Y 418.909,Z 731.954,A -85,B 0,C 180,E1 -10001.123,E2 -10001.123} C_VEL
LIN {X 0,Y 419.461,Z 723.903,A -85,B 0,C 180,E1 -10002.334,E2 -10002.334} C_VEL
LIN {X 0,Y 420.287,Z 714.069,A -85,B 0,C 180,E1 -10003.538,E2 -10003.538} C_VEL
LIN {X 0,Y 420.931,Z 703.02,A -85,B 0,C 180,E1 -10004.626,E2 -10004.626} C_VEL
LIN {X 0,Y 421.628,Z 692.176,A -85,B 0,C 180,E1 -10005.467,E2 -10005.467} C_VEL
LIN {X 0,Y 422.283,Z 680.191,A -85,B 0,C 180,E1 -10006.186,E2 -10006.186} C_VEL
LIN {X 0,Y 422.749,Z 667.924,A -85,B 0,C 180,E1 -10006.726,E2 -10006.726} C_VEL
LIN {X 0,Y 423.12,Z 655.31,A -85,B 0,C 180,E1 -10007.084,E2 -10007.084} C_VEL
LIN {X 0,Y 423.993,Z 570.569,A -85,B 0,C 180,E1 -10008.539,E2 -10008.539} C_VEL
LIN {X 0,Y 420.075,Z 550.932,A -85,B 0,C 180,E1 -10009.089,E2 -10009.089} C_VEL
LIN {X 0,Y 420.041,Z 549.548,A -85,B 0,C 180,E1 -10009.302,E2 -10009.302} C_VEL
LIN {X 0,Y 420.265,Z 543.185,A -85,B 0,C 180,E1 -10010.814,E2 -10010.814} C_VEL
LIN {X 0,Y 418.347,Z 532.676,A -85,B 0,C 180,E1 -10013.514,E2 -10013.514} C_VEL
LIN {X 0,Y 418.288,Z 532.377,A -85,B 0,C 180,E1 -10013.78,E2 -10013.78} C_VEL
LIN {X 0,Y 418.309,Z 532.377,A -85,B 0,C 180,E1 -10017.069,E2 -10017.069} C_VEL
LIN {X 0,Y 418.243,Z 532.381,A -85,B 0,C 180,E1 -10020.271,E2 -10020.271} C_VEL
LIN {X 0,Y 418.247,Z 532.389,A -85,B 0,C 180,E1 -10023.676,E2 -10023.676} C_VEL
LIN {X 0,Y 418.243,Z 532.386,A -85,B 0,C 180,E1 -10027.222,E2 -10027.222} C_VEL
LIN {X 0,Y 418.252,Z 532.379,A -85,B 0,C 180,E1 -10029.68,E2 -10029.68} C_VEL
LIN {X 0,Y 418.229,Z 532.386,A -85,B 0,C 180,E1 -10032.321,E2 -10032.321} C_VEL
LIN {X 0,Y 418.234,Z 532.377,A -85,B 0,C 180,E1 -10035.108,E2 -10035.108} C_VEL
LIN {X 0,Y 418.251,Z 532.386,A -85,B 0,C 180,E1 -10037.768,E2 -10037.768} C_VEL
LIN {X 0,Y 418.264,Z 532.372,A -85,B 0,C 180,E1 -10040.616,E2 -10040.616} C_VEL
LIN {X 0,Y 418.243,Z 532.385,A -85,B 0,C 180,E1 -10043.976,E2 -10043.976} C_VEL
LIN {X 0,Y 418.252,Z 532.385,A -85,B 0,C 180,E1 -10047.155,E2 -10047.155} C_VEL
LIN {X 0,Y 418.268,Z 532.381,A -85,B 0,C 180,E1 -10050.838,E2 -10050.838} C_VEL
LIN {X 0,Y 418.264,Z 532.382,A -85,B 0,C 180,E1 -10054.095,E2 -10054.095} C_VEL
LIN {X 0,Y 418.231,Z 532.385,A -85,B 0,C 180,E1 -10057.263,E2 -10057.263} C_VEL
LIN {X 0,Y 418.276,Z 532.379,A -85,B 0,C 180,E1 -10060.364,E2 -10060.364} C_VEL
LIN {X 0,Y 418.309,Z 532.372,A -85,B 0,C 180,E1 -10063.404,E2 -10063.404} C_VEL
LIN {X 0,Y 418.338,Z 532.372,A -85,B 0,C 180,E1 -10066.999,E2 -10066.999} C_VEL
LIN {X 0,Y 418.334,Z 532.364,A -85,B 0,C 180,E1 -10070.328,E2 -10070.328} C_VEL
LIN {X 0,Y 418.486,Z 532.356,A -85,B 0,C 180,E1 -10073.249,E2 -10073.249} C_VEL
LIN {X 0,Y 418.334,Z 532.374,A -85,B 0,C 180,E1 -10075.181,E2 -10075.181} C_VEL
LIN {X 0,Y 418.537,Z 532.346,A -85,B 0,C 180,E1 -10078.075,E2 -10078.075} C_VEL
LIN {X 0,Y 418.667,Z 532.333,A -85,B 0,C 180,E1 -10080,E2 -10080} C_VEL
LIN {X 0,Y 418.504,Z 532.347,A -85,B 0,C 180,E1 -10082.888,E2 -10082.888} C_VEL
LIN {X 0,Y 418.522,Z 532.353,A -85,B 0,C 180,E1 -10085.783,E2 -10085.783} C_VEL
LIN {X 0,Y 418.393,Z 532.362,A -85,B 0,C 180,E1 -10088.695,E2 -10088.695} C_VEL
LIN {X 0,Y 418.324,Z 532.374,A -85,B 0,C 180,E1 -10091.631,E2 -10091.631} C_VEL
LIN {X 0,Y 418.298,Z 532.374,A -85,B 0,C 180,E1 -10094.597,E2 -10094.597} C_VEL
LIN {X 0,Y 418.281,Z 532.38,A -85,B 0,C 180,E1 -10097.604,E2 -10097.604} C_VEL
LIN {X 0,Y 418.253,Z 532.38,A -85,B 0,C 180,E1 -10100.663,E2 -10100.663} C_VEL
LIN {X 0,Y 418.281,Z 532.384,A -85,B 0,C 180,E1 -10103.782,E2 -10103.782} C_VEL
LIN {X 0,Y 418.303,Z 532.372,A -85,B 0,C 180,E1 -10107.071,E2 -10107.071} C_VEL
LIN {X 0,Y 418.238,Z 532.382,A -85,B 0,C 180,E1 -10110.273,E2 -10110.273} C_VEL
LIN {X 0,Y 418.243,Z 532.388,A -85,B 0,C 180,E1 -10113.678,E2 -10113.678} C_VEL
LIN {X 0,Y 418.24,Z 532.372,A -85,B 0,C 180,E1 -10117.224,E2 -10117.224} C_VEL
LIN {X 0,Y 418.25,Z 532.39,A -85,B 0,C 180,E1 -10119.682,E2 -10119.682} C_VEL
LIN {X 0,Y 418.224,Z 532.377,A -85,B 0,C 180,E1 -10122.322,E2 -10122.322} C_VEL
LIN {X 0,Y 418.255,Z 532.384,A -85,B 0,C 180,E1 -10125.113,E2 -10125.113} C_VEL
LIN {X 0,Y 418.288,Z 532.378,A -85,B 0,C 180,E1 -10127.774,E2 -10127.774} C_VEL
LIN {X 0,Y 418.262,Z 532.367,A -85,B 0,C 180,E1 -10131.561,E2 -10131.561} C_VEL
LIN {X 0,Y 418.257,Z 532.386,A -85,B 0,C 180,E1 -10135.16,E2 -10135.16} C_VEL
LIN {X 0,Y 418.243,Z 532.348,A -85,B 0,C 180,E1 -10137.473,E2 -10137.473} C_VEL
LIN {X 0,Y 418.267,Z 532.365,A -85,B 0,C 180,E1 -10140.896,E2 -10140.896} C_VEL
LIN {X 0,Y 418.352,Z 532.554,A -85,B 0,C 180,E1 -10142.528,E2 -10142.528} C_VEL
LIN {X 0,Y 420.855,Z 544.96,A -85,B 0,C 180,E1 -10145.325,E2 -10145.325} C_VEL
LIN {X 0,Y 421.335,Z 548.765,A -85,B 0,C 180,E1 -10146.141,E2 -10146.141} C_VEL
LIN {X 0,Y 420.308,Z 563.854,A -85,B 0,C 180,E1 -10149.188,E2 -10149.188} C_VEL
LIN {X 0,Y 419.802,Z 572.715,A -85,B 0,C 180,E1 -10150.916,E2 -10150.916} C_VEL
LIN {X 0,Y 423.715,Z 597.05,A -85,B 0,C 180,E1 -10151.552,E2 -10151.552} C_VEL
LIN {X 0,Y 422.896,Z 680.761,A -85,B 0,C 180,E1 -10153,E2 -10153} C_VEL
LIN {X 0,Y 422.394,Z 693.994,A -85,B 0,C 180,E1 -10153.415,E2 -10153.415} C_VEL
LIN {X 0,Y 421.796,Z 706.144,A -85,B 0,C 180,E1 -10153.981,E2 -10153.981} C_VEL
LIN {X 0,Y 421.049,Z 718.413,A -85,B 0,C 180,E1 -10154.759,E2 -10154.759} C_VEL
LIN {X 0,Y 420.251,Z 729.597,A -85,B 0,C 180,E1 -10155.682,E2 -10155.682} C_VEL
LIN {X 0,Y 419.538,Z 740.445,A -85,B 0,C 180,E1 -10156.807,E2 -10156.807} C_VEL
LIN {X 0,Y 418.921,Z 748.984,A -85,B 0,C 180,E1 -10157.896,E2 -10157.896} C_VEL
LIN {X 0,Y 418.316,Z 756.861,A -85,B 0,C 180,E1 -10159.106,E2 -10159.106} C_VEL
LIN {X 0,Y 417.794,Z 764.558,A -85,B 0,C 180,E1 -10160.561,E2 -10160.561} C_VEL
LIN {X 0,Y 417.384,Z 771.654,A -85,B 0,C 180,E1 -10162.259,E2 -10162.259} C_VEL
LIN {X 0,Y 417.146,Z 776.432,A -85,B 0,C 180,E1 -10163.733,E2 -10163.733} C_VEL
LIN {X 0,Y 417.113,Z 779.991,A -85,B 0,C 180,E1 -10165.168,E2 -10165.168} C_VEL
LIN {X 0,Y 417.016,Z 781.852,A -85,B 0,C 180,E1 -10166.136,E2 -10166.136} C_VEL
LIN {X 0,Y 417.029,Z 783.248,A -85,B 0,C 180,E1 -10167.103,E2 -10167.103} C_VEL
LIN {X 0,Y 417.056,Z 784.244,A -85,B 0,C 180,E1 -10168.069,E2 -10168.069} C_VEL
LIN {X 0,Y 417.004,Z 785.193,A -85,B 0,C 180,E1 -10170.001,E2 -10170.001} C_VEL
LIN {X 0,Y 417.01,Z 784.983,A -85,B 0,C 180,E1 -10170.967,E2 -10170.967} C_VEL
LIN {X 0,Y 417.029,Z 783.239,A -85,B 0,C 180,E1 -10172.899,E2 -10172.899} C_VEL
LIN {X 0,Y 417.017,Z 781.84,A -85,B 0,C 180,E1 -10173.866,E2 -10173.866} C_VEL
LIN {X 0,Y 417.132,Z 778.905,A -85,B 0,C 180,E1 -10175.318,E2 -10175.318} C_VEL
LIN {X 0,Y 417.236,Z 774.929,A -85,B 0,C 180,E1 -10176.772,E2 -10176.772} C_VEL
LIN {X 0,Y 417.545,Z 768.812,A -85,B 0,C 180,E1 -10178.47,E2 -10178.47} C_VEL
LIN {X 0,Y 417.946,Z 762.131,A -85,B 0,C 180,E1 -10179.926,E2 -10179.926} C_VEL
LIN {X 0,Y 418.522,Z 753.844,A -85,B 0,C 180,E1 -10181.381,E2 -10181.381} C_VEL
LIN {X 0,Y 419.208,Z 745.352,A -85,B 0,C 180,E1 -10182.589,E2 -10182.589} C_VEL
LIN {X 0,Y 419.911,Z 734.725,A -85,B 0,C 180,E1 -10183.813,E2 -10183.813} C_VEL
LIN {X 0,Y 420.703,Z 723.044,A -85,B 0,C 180,E1 -10184.884,E2 -10184.884} C_VEL
LIN {X 0,Y 421.466,Z 711.172,A -85,B 0,C 180,E1 -10185.723,E2 -10185.723} C_VEL
LIN {X 0,Y 422.151,Z 698.821,A -85,B 0,C 180,E1 -10186.379,E2 -10186.379} C_VEL
LIN {X 0,Y 422.702,Z 686.124,A -85,B 0,C 180,E1 -10186.854,E2 -10186.854} C_VEL
LIN {X 0,Y 423.037,Z 672.816,A -85,B 0,C 180,E1 -10187.151,E2 -10187.151} C_VEL
LIN {X 0,Y 423.692,Z 597.321,A -85,B 0,C 180,E1 -10188.439,E2 -10188.439} C_VEL
LIN {X 0,Y 419.8,Z 572.9,A -85,B 0,C 180,E1 -10189.063,E2 -10189.063} C_VEL
LIN {X 0,Y 419.923,Z 570.067,A -85,B 0,C 180,E1 -10189.557,E2 -10189.557} C_VEL
LIN {X 0,Y 421.231,Z 550.903,A -85,B 0,C 180,E1 -10193.416,E2 -10193.416} C_VEL
LIN {X 0,Y 421.249,Z 547.455,A -85,B 0,C 180,E1 -10194.127,E2 -10194.127} C_VEL
LIN {X 0,Y 419.09,Z 536.015,A -85,B 0,C 180,E1 -10196.654,E2 -10196.654} C_VEL
LIN {X 0,Y 418.357,Z 532.411,A -85,B 0,C 180,E1 -10197.539,E2 -10197.539} C_VEL
LIN {X 0,Y 418.243,Z 532.387,A -85,B 0,C 180,E1 -10201.02,E2 -10201.02} C_VEL
LIN {X 0,Y 418.253,Z 532.385,A -85,B 0,C 180,E1 -10203.678,E2 -10203.678} C_VEL
LIN {X 0,Y 418.244,Z 532.384,A -85,B 0,C 180,E1 -10207.225,E2 -10207.225} C_VEL
LIN {X 0,Y 418.252,Z 532.386,A -85,B 0,C 180,E1 -10209.683,E2 -10209.683} C_VEL
LIN {X 0,Y 418.234,Z 532.387,A -85,B 0,C 180,E1 -10212.322,E2 -10212.322} C_VEL
LIN {X 0,Y 418.24,Z 532.387,A -85,B 0,C 180,E1 -10215.109,E2 -10215.109} C_VEL
LIN {X 0,Y 418.244,Z 532.387,A -85,B 0,C 180,E1 -10217.767,E2 -10217.767} C_VEL
LIN {X 0,Y 418.261,Z 532.386,A -85,B 0,C 180,E1 -10221.559,E2 -10221.559} C_VEL
LIN {X 0,Y 418.264,Z 532.384,A -85,B 0,C 180,E1 -10225.159,E2 -10225.159} C_VEL
LIN {X 0,Y 418.249,Z 532.389,A -85,B 0,C 180,E1 -10227.472,E2 -10227.472} C_VEL
LIN {X 0,Y 418.303,Z 532.612,A -85,B 0,C 180,E1 -10230.133,E2 -10230.133} C_VEL
LIN {X 0,Y 420.839,Z 541.861,A -85,B 0,C 180,E1 -10231.85,E2 -10231.85} C_VEL
LIN {X 0,Y 422.499,Z 550.28,A -85,B 0,C 180,E1 -10233.312,E2 -10233.312} C_VEL
LIN {X 0,Y 422.445,Z 556.998,A -85,B 0,C 180,E1 -10234.371,E2 -10234.371} C_VEL
LIN {X 0,Y 421.502,Z 576.914,A -85,B 0,C 180,E1 -10237.45,E2 -10237.45} C_VEL
LIN {X 0,Y 420.61,Z 598.118,A -85,B 0,C 180,E1 -10240.731,E2 -10240.731} C_VEL
LIN {X 0,Y 419.725,Z 620.486,A -85,B 0,C 180,E1 -10244.211,E2 -10244.211} C_VEL
LIN {X 0,Y 419.362,Z 631.822,A -85,B 0,C 180,E1 -10245.936,E2 -10245.936} C_VEL
LIN {X 0,Y 421.142,Z 647.111,A -85,B 0,C 180,E1 -10246.379,E2 -10246.379} C_VEL
LIN {X 0,Y 420.203,Z 703.803,A -85,B 0,C 180,E1 -10247.595,E2 -10247.595} C_VEL
LIN {X 0,Y 419.886,Z 714.433,A -85,B 0,C 180,E1 -10247.984,E2 -10247.984} C_VEL
LIN {X 0,Y 419.55,Z 724.655,A -85,B 0,C 180,E1 -10248.526,E2 -10248.526} C_VEL
LIN {X 0,Y 419.123,Z 734.447,A -85,B 0,C 180,E1 -10249.249,E2 -10249.249} C_VEL
LIN {X 0,Y 418.771,Z 742.195,A -85,B 0,C 180,E1 -10249.973,E2 -10249.973} C_VEL
LIN {X 0,Y 418.361,Z 749.577,A -85,B 0,C 180,E1 -10250.817,E2 -10250.817} C_VEL
LIN {X 0,Y 417.898,Z 757.906,A -85,B 0,C 180,E1 -10252.025,E2 -10252.025} C_VEL
LIN {X 0,Y 417.603,Z 764.335,A -85,B 0,C 180,E1 -10253.235,E2 -10253.235} C_VEL
LIN {X 0,Y 417.36,Z 770.27,A -85,B 0,C 180,E1 -10254.686,E2 -10254.686} C_VEL
LIN {X 0,Y 417.174,Z 773.253,A -85,B 0,C 180,E1 -10255.652,E2 -10255.652} C_VEL
LIN {X 0,Y 417.119,Z 776.391,A -85,B 0,C 180,E1 -10257.103,E2 -10257.103} C_VEL
LIN {X 0,Y 417.064,Z 777.764,A -85,B 0,C 180,E1 -10258.069,E2 -10258.069} C_VEL
LIN {X 0,Y 416.992,Z 778.559,A -85,B 0,C 180,E1 -10259.034,E2 -10259.034} C_VEL
LIN {X 0,Y 416.982,Z 778.786,A -85,B 0,C 180,E1 -10260,E2 -10260} C_VEL
LIN {X 0,Y 416.993,Z 778.421,A -85,B 0,C 180,E1 -10260.966,E2 -10260.966} C_VEL
LIN {X 0,Y 417.061,Z 777.454,A -85,B 0,C 180,E1 -10261.931,E2 -10261.931} C_VEL
LIN {X 0,Y 417.113,Z 774.862,A -85,B 0,C 180,E1 -10263.381,E2 -10263.381} C_VEL
LIN {X 0,Y 417.217,Z 770.848,A -85,B 0,C 180,E1 -10264.832,E2 -10264.832} C_VEL
LIN {X 0,Y 417.366,Z 765.358,A -85,B 0,C 180,E1 -10266.251,E2 -10266.251} C_VEL
LIN {X 0,Y 417.608,Z 760.313,A -85,B 0,C 180,E1 -10267.251,E2 -10267.251} C_VEL
LIN {X 0,Y 417.821,Z 754.329,A -85,B 0,C 180,E1 -10268.22,E2 -10268.22} C_VEL
LIN {X 0,Y 418.138,Z 746.991,A -85,B 0,C 180,E1 -10269.188,E2 -10269.188} C_VEL
LIN {X 0,Y 418.571,Z 737.748,A -85,B 0,C 180,E1 -10270.154,E2 -10270.154} C_VEL
LIN {X 0,Y 418.953,Z 728.689,A -85,B 0,C 180,E1 -10270.878,E2 -10270.878} C_VEL
LIN {X 0,Y 419.227,Z 718.905,A -85,B 0,C 180,E1 -10271.483,E2 -10271.483} C_VEL
LIN {X 0,Y 419.548,Z 707.653,A -85,B 0,C 180,E1 -10271.964,E2 -10271.964} C_VEL
LIN {X 0,Y 419.688,Z 695.952,A -85,B 0,C 180,E1 -10272.267,E2 -10272.267} C_VEL
LIN {X 0,Y 420.2,Z 644.875,A -85,B 0,C 180,E1 -10273.293,E2 -10273.293} C_VEL
LIN {X 0,Y 418.806,Z 631.645,A -85,B 0,C 180,E1 -10273.619,E2 -10273.619} C_VEL
LIN {X 0,Y 419.51,Z 611.544,A -85,B 0,C 180,E1 -10276.733,E2 -10276.733} C_VEL
LIN {X 0,Y 420.4,Z 588.881,A -85,B 0,C 180,E1 -10280.297,E2 -10280.297} C_VEL
LIN {X 0,Y 421.346,Z 566.315,A -85,B 0,C 180,E1 -10283.859,E2 -10283.859} C_VEL
LIN {X 0,Y 422.055,Z 551.488,A -85,B 0,C 180,E1 -10286.204,E2 -10286.204} C_VEL
LIN {X 0,Y 420.745,Z 543.905,A -85,B 0,C 180,E1 -10287.482,E2 -10287.482} C_VEL
LIN {X 0,Y 418.327,Z 532.5,A -85,B 0,C 180,E1 -10289.485,E2 -10289.485} C_VEL
LIN {X 0,Y 418.262,Z 532.386,A -85,B 0,C 180,E1 -10292.844,E2 -10292.844} C_VEL
LIN {X 0,Y 418.253,Z 532.388,A -85,B 0,C 180,E1 -10296.239,E2 -10296.239} C_VEL
LIN {X 0,Y 418.254,Z 532.38,A -85,B 0,C 180,E1 -10299.682,E2 -10299.682} C_VEL
LIN {X 0,Y 418.234,Z 532.362,A -85,B 0,C 180,E1 -10302.321,E2 -10302.321} C_VEL
LIN {X 0,Y 418.244,Z 532.382,A -85,B 0,C 180,E1 -10305.109,E2 -10305.109} C_VEL
LIN {X 0,Y 418.261,Z 532.382,A -85,B 0,C 180,E1 -10307.769,E2 -10307.769} C_VEL
LIN {X 0,Y 418.255,Z 532.374,A -85,B 0,C 180,E1 -10311.558,E2 -10311.558} C_VEL
LIN {X 0,Y 418.264,Z 532.375,A -85,B 0,C 180,E1 -10315.159,E2 -10315.159} C_VEL
LIN {X 0,Y 418.25,Z 532.384,A -85,B 0,C 180,E1 -10317.472,E2 -10317.472} C_VEL
LIN {X 0,Y 418.273,Z 532.382,A -85,B 0,C 180,E1 -10320.895,E2 -10320.895} C_VEL
LIN {X 0,Y 418.273,Z 532.383,A -85,B 0,C 180,E1 -10324.095,E2 -10324.095} C_VEL
LIN {X 0,Y 418.327,Z 532.586,A -85,B 0,C 180,E1 -10326.549,E2 -10326.549} C_VEL
LIN {X 0,Y 420.257,Z 542.777,A -85,B 0,C 180,E1 -10329.183,E2 -10329.183} C_VEL
LIN {X 0,Y 420.003,Z 550.129,A -85,B 0,C 180,E1 -10330.91,E2 -10330.91} C_VEL
LIN {X 0,Y 420.102,Z 551.332,A -85,B 0,C 180,E1 -10331.025,E2 -10331.025} C_VEL
LIN {X 0,Y 424.054,Z 570.829,A -85,B 0,C 180,E1 -10331.564,E2 -10331.564} C_VEL
LIN {X 0,Y 423.006,Z 657.826,A -85,B 0,C 180,E1 -10333.065,E2 -10333.065} C_VEL
LIN {X 0,Y 422.816,Z 665.53,A -85,B 0,C 180,E1 -10333.289,E2 -10333.289} C_VEL
LIN {X 0,Y 422.01,Z 671.241,A -85,B 0,C 180,E1 -10333.467,E2 -10333.467} C_VEL
LIN {X 0,Y 418.92,Z 680.414,A -85,B 0,C 180,E1 -10333.766,E2 -10333.766} C_VEL
LIN {X 0,Y 415.679,Z 689.289,A -85,B 0,C 180,E1 -10334.171,E2 -10334.171} C_VEL
LIN {X 0,Y 414.642,Z 694.528,A -85,B 0,C 180,E1 -10334.517,E2 -10334.517} C_VEL
LIN {X 0,Y 413.936,Z 705.354,A -85,B 0,C 180,E1 -10335.416,E2 -10335.416} C_VEL
LIN {X 0,Y 413.172,Z 716.641,A -85,B 0,C 180,E1 -10336.599,E2 -10336.599} C_VEL
LIN {X 0,Y 412.458,Z 725.188,A -85,B 0,C 180,E1 -10337.701,E2 -10337.701} C_VEL
LIN {X 0,Y 411.849,Z 733.06,A -85,B 0,C 180,E1 -10338.931,E2 -10338.931} C_VEL
LIN {X 0,Y 411.224,Z 740.754,A -85,B 0,C 180,E1 -10340.407,E2 -10340.407} C_VEL
LIN {X 0,Y 410.611,Z 747.816,A -85,B 0,C 180,E1 -10342.129,E2 -10342.129} C_VEL
LIN {X 0,Y 410.394,Z 752.599,A -85,B 0,C 180,E1 -10343.637,E2 -10343.637} C_VEL
LIN {X 0,Y 410.165,Z 756.112,A -85,B 0,C 180,E1 -10345.084,E2 -10345.084} C_VEL
LIN {X 0,Y 410.058,Z 757.971,A -85,B 0,C 180,E1 -10346.068,E2 -10346.068} C_VEL
LIN {X 0,Y 410.061,Z 759.371,A -85,B 0,C 180,E1 -10347.052,E2 -10347.052} C_VEL
LIN {X 0,Y 410.013,Z 760.368,A -85,B 0,C 180,E1 -10348.035,E2 -10348.035} C_VEL
LIN {X 0,Y 409.927,Z 761.219,A -85,B 0,C 180,E1 -10349.999,E2 -10349.999} C_VEL
LIN {X 0,Y 409.939,Z 761.032,A -85,B 0,C 180,E1 -10350.981,E2 -10350.981} C_VEL
LIN {X 0,Y 410.012,Z 760.448,A -85,B 0,C 180,E1 -10351.964,E2 -10351.964} C_VEL
LIN {X 0,Y 410.056,Z 759.483,A -85,B 0,C 180,E1 -10352.946,E2 -10352.946} C_VEL
LIN {X 0,Y 410.046,Z 758.131,A -85,B 0,C 180,E1 -10353.93,E2 -10353.93} C_VEL
LIN {X 0,Y 410.267,Z 755.263,A -85,B 0,C 180,E1 -10355.405,E2 -10355.405} C_VEL
LIN {X 0,Y 410.462,Z 751.377,A -85,B 0,C 180,E1 -10356.883,E2 -10356.883} C_VEL
LIN {X 0,Y 410.756,Z 746.368,A -85,B 0,C 180,E1 -10358.361,E2 -10358.361} C_VEL
LIN {X 0,Y 411.302,Z 740.058,A -85,B 0,C 180,E1 -10359.838,E2 -10359.838} C_VEL
LIN {X 0,Y 411.931,Z 732.156,A -85,B 0,C 180,E1 -10361.314,E2 -10361.314} C_VEL
LIN {X 0,Y 412.539,Z 724.104,A -85,B 0,C 180,E1 -10362.544,E2 -10362.544} C_VEL
LIN {X 0,Y 413.399,Z 714.269,A -85,B 0,C 180,E1 -10363.768,E2 -10363.768} C_VEL
LIN {X 0,Y 414.058,Z 703.22,A -85,B 0,C 180,E1 -10364.875,E2 -10364.875} C_VEL
LIN {X 0,Y 414.787,Z 692.375,A -85,B 0,C 180,E1 -10365.729,E2 -10365.729} C_VEL
LIN {X 0,Y 415.493,Z 680.387,A -85,B 0,C 180,E1 -10366.458,E2 -10366.458} C_VEL
LIN {X 0,Y 415.978,Z 668.116,A -85,B 0,C 180,E1 -10367.006,E2 -10367.006} C_VEL
LIN {X 0,Y 416.36,Z 655.492,A -85,B 0,C 180,E1 -10367.37,E2 -10367.37} C_VEL
LIN {X 0,Y 417.221,Z 571.282,A -85,B 0,C 180,E1 -10368.841,E2 -10368.841} C_VEL
LIN {X 0,Y 413.18,Z 551.195,A -85,B 0,C 180,E1 -10369.416,E2 -10369.416} C_VEL
LIN {X 0,Y 413.119,Z 550.417,A -85,B 0,C 180,E1 -10369.502,E2 -10369.502} C_VEL
LIN {X 0,Y 413.306,Z 544.437,A -85,B 0,C 180,E1 -10370.921,E2 -10370.921} C_VEL
LIN {X 0,Y 411.382,Z 533.886,A -85,B 0,C 180,E1 -10373.669,E2 -10373.669} C_VEL
LIN {X 0,Y 411.248,Z 533.269,A -85,B 0,C 180,E1 -10373.945,E2 -10373.945} C_VEL
LIN {X 0,Y 411.258,Z 533.26,A -85,B 0,C 180,E1 -10377.477,E2 -10377.477} C_VEL
LIN {X 0,Y 411.188,Z 533.262,A -85,B 0,C 180,E1 -10380.846,E2 -10380.846} C_VEL
LIN {X 0,Y 411.204,Z 533.263,A -85,B 0,C 180,E1 -10384.332,E2 -10384.332} C_VEL
LIN {X 0,Y 411.198,Z 533.263,A -85,B 0,C 180,E1 -10387.972,E2 -10387.972} C_VEL
LIN {X 0,Y 411.19,Z 533.263,A -85,B 0,C 180,E1 -10391.232,E2 -10391.232} C_VEL
LIN {X 0,Y 411.175,Z 533.256,A -85,B 0,C 180,E1 -10394.489,E2 -10394.489} C_VEL
LIN {X 0,Y 411.194,Z 533.262,A -85,B 0,C 180,E1 -10398.196,E2 -10398.196} C_VEL
LIN {X 0,Y 411.227,Z 533.248,A -85,B 0,C 180,E1 -10400.777,E2 -10400.777} C_VEL
LIN {X 0,Y 411.196,Z 533.261,A -85,B 0,C 180,E1 -10404.471,E2 -10404.471} C_VEL
LIN {X 0,Y 411.162,Z 533.265,A -85,B 0,C 180,E1 -10408.002,E2 -10408.002} C_VEL
LIN {X 0,Y 411.218,Z 533.26,A -85,B 0,C 180,E1 -10411.41,E2 -10411.41} C_VEL
LIN {X 0,Y 411.23,Z 533.257,A -85,B 0,C 180,E1 -10414.706,E2 -10414.706} C_VEL
LIN {X 0,Y 411.198,Z 533.258,A -85,B 0,C 180,E1 -10417.913,E2 -10417.913} C_VEL
LIN {X 0,Y 411.218,Z 533.26,A -85,B 0,C 180,E1 -10421.051,E2 -10421.051} C_VEL
LIN {X 0,Y 411.247,Z 533.25,A -85,B 0,C 180,E1 -10424.131,E2 -10424.131} C_VEL
LIN {X 0,Y 411.295,Z 533.251,A -85,B 0,C 180,E1 -10427.165,E2 -10427.165} C_VEL
LIN {X 0,Y 411.286,Z 533.242,A -85,B 0,C 180,E1 -10430.161,E2 -10430.161} C_VEL
LIN {X 0,Y 411.453,Z 533.231,A -85,B 0,C 180,E1 -10433.133,E2 -10433.133} C_VEL
LIN {X 0,Y 411.305,Z 533.249,A -85,B 0,C 180,E1 -10435.099,E2 -10435.099} C_VEL
LIN {X 0,Y 411.506,Z 533.222,A -85,B 0,C 180,E1 -10438.042,E2 -10438.042} C_VEL
LIN {X 0,Y 411.636,Z 533.209,A -85,B 0,C 180,E1 -10440,E2 -10440} C_VEL
LIN {X 0,Y 411.46,Z 533.224,A -85,B 0,C 180,E1 -10442.937,E2 -10442.937} C_VEL
LIN {X 0,Y 411.481,Z 533.229,A -85,B 0,C 180,E1 -10445.882,E2 -10445.882} C_VEL
LIN {X 0,Y 411.474,Z 533.228,A -85,B 0,C 180,E1 -10447.853,E2 -10447.853} C_VEL
LIN {X 0,Y 411.291,Z 533.253,A -85,B 0,C 180,E1 -10451.833,E2 -10451.833} C_VEL
LIN {X 0,Y 411.255,Z 533.252,A -85,B 0,C 180,E1 -10454.853,E2 -10454.853} C_VEL
LIN {X 0,Y 411.245,Z 533.259,A -85,B 0,C 180,E1 -10457.915,E2 -10457.915} C_VEL
LIN {X 0,Y 411.195,Z 533.26,A -85,B 0,C 180,E1 -10461.034,E2 -10461.034} C_VEL
LIN {X 0,Y 411.22,Z 533.26,A -85,B 0,C 180,E1 -10464.216,E2 -10464.216} C_VEL
LIN {X 0,Y 411.252,Z 533.254,A -85,B 0,C 180,E1 -10467.478,E2 -10467.478} C_VEL
LIN {X 0,Y 411.184,Z 533.26,A -85,B 0,C 180,E1 -10470.848,E2 -10470.848} C_VEL
LIN {X 0,Y 411.2,Z 533.258,A -85,B 0,C 180,E1 -10474.334,E2 -10474.334} C_VEL
LIN {X 0,Y 411.195,Z 533.26,A -85,B 0,C 180,E1 -10477.974,E2 -10477.974} C_VEL
LIN {X 0,Y 411.178,Z 533.263,A -85,B 0,C 180,E1 -10480.505,E2 -10480.505} C_VEL
LIN {X 0,Y 411.169,Z 533.257,A -85,B 0,C 180,E1 -10483.134,E2 -10483.134} C_VEL
LIN {X 0,Y 411.223,Z 533.258,A -85,B 0,C 180,E1 -10485.873,E2 -10485.873} C_VEL
LIN {X 0,Y 411.206,Z 533.261,A -85,B 0,C 180,E1 -10488.765,E2 -10488.765} C_VEL
LIN {X 0,Y 411.201,Z 533.243,A -85,B 0,C 180,E1 -10492.028,E2 -10492.028} C_VEL
LIN {X 0,Y 411.203,Z 533.26,A -85,B 0,C 180,E1 -10495.668,E2 -10495.668} C_VEL
LIN {X 0,Y 411.187,Z 533.212,A -85,B 0,C 180,E1 -10499.153,E2 -10499.153} C_VEL
LIN {X 0,Y 411.305,Z 533.44,A -85,B 0,C 180,E1 -10502.251,E2 -10502.251} C_VEL
LIN {X 0,Y 413.867,Z 546.036,A -85,B 0,C 180,E1 -10505.148,E2 -10505.148} C_VEL
LIN {X 0,Y 414.399,Z 549.84,A -85,B 0,C 180,E1 -10505.983,E2 -10505.983} C_VEL
LIN {X 0,Y 413.263,Z 565.894,A -85,B 0,C 180,E1 -10509.283,E2 -10509.283} C_VEL
LIN {X 0,Y 412.873,Z 572.513,A -85,B 0,C 180,E1 -10510.583,E2 -10510.583} C_VEL
LIN {X 0,Y 417.033,Z 598.475,A -85,B 0,C 180,E1 -10511.274,E2 -10511.274} C_VEL
LIN {X 0,Y 416.118,Z 680.568,A -85,B 0,C 180,E1 -10512.715,E2 -10512.715} C_VEL
LIN {X 0,Y 415.545,Z 693.796,A -85,B 0,C 180,E1 -10513.134,E2 -10513.134} C_VEL
LIN {X 0,Y 414.909,Z 707.065,A -85,B 0,C 180,E1 -10513.771,E2 -10513.771} C_VEL
LIN {X 0,Y 414.196,Z 718.213,A -85,B 0,C 180,E1 -10514.501,E2 -10514.501} C_VEL
LIN {X 0,Y 413.331,Z 729.885,A -85,B 0,C 180,E1 -10515.484,E2 -10515.484} C_VEL
LIN {X 0,Y 412.591,Z 740.242,A -85,B 0,C 180,E1 -10516.581,E2 -10516.581} C_VEL
LIN {X 0,Y 411.954,Z 748.781,A -85,B 0,C 180,E1 -10517.688,E2 -10517.688} C_VEL
LIN {X 0,Y 411.322,Z 756.657,A -85,B 0,C 180,E1 -10518.919,E2 -10518.919} C_VEL
LIN {X 0,Y 410.762,Z 764.353,A -85,B 0,C 180,E1 -10520.398,E2 -10520.398} C_VEL
LIN {X 0,Y 410.341,Z 771.45,A -85,B 0,C 180,E1 -10522.126,E2 -10522.126} C_VEL
LIN {X 0,Y 410.043,Z 776.658,A -85,B 0,C 180,E1 -10523.775,E2 -10523.775} C_VEL
LIN {X 0,Y 410.025,Z 779.786,A -85,B 0,C 180,E1 -10525.085,E2 -10525.085} C_VEL
LIN {X 0,Y 409.935,Z 781.648,A -85,B 0,C 180,E1 -10526.069,E2 -10526.069} C_VEL
LIN {X 0,Y 409.966,Z 784.04,A -85,B 0,C 180,E1 -10528.036,E2 -10528.036} C_VEL
LIN {X 0,Y 409.926,Z 785.115,A -85,B 0,C 180,E1 -10530.001,E2 -10530.001} C_VEL
LIN {X 0,Y 409.935,Z 784.922,A -85,B 0,C 180,E1 -10530.983,E2 -10530.983} C_VEL
LIN {X 0,Y 409.967,Z 784.165,A -85,B 0,C 180,E1 -10531.966,E2 -10531.966} C_VEL
LIN {X 0,Y 409.935,Z 781.635,A -85,B 0,C 180,E1 -10533.933,E2 -10533.933} C_VEL
LIN {X 0,Y 410.028,Z 778.698,A -85,B 0,C 180,E1 -10535.41,E2 -10535.41} C_VEL
LIN {X 0,Y 410.169,Z 774.723,A -85,B 0,C 180,E1 -10536.89,E2 -10536.89} C_VEL
LIN {X 0,Y 410.493,Z 768.605,A -85,B 0,C 180,E1 -10538.617,E2 -10538.617} C_VEL
LIN {X 0,Y 410.939,Z 761.924,A -85,B 0,C 180,E1 -10540.097,E2 -10540.097} C_VEL
LIN {X 0,Y 411.543,Z 753.637,A -85,B 0,C 180,E1 -10541.576,E2 -10541.576} C_VEL
LIN {X 0,Y 412.253,Z 745.144,A -85,B 0,C 180,E1 -10542.805,E2 -10542.805} C_VEL
LIN {X 0,Y 412.984,Z 734.337,A -85,B 0,C 180,E1 -10544.068,E2 -10544.068} C_VEL
LIN {X 0,Y 413.831,Z 722.835,A -85,B 0,C 180,E1 -10545.137,E2 -10545.137} C_VEL
LIN {X 0,Y 414.641,Z 710.963,A -85,B 0,C 180,E1 -10545.988,E2 -10545.988} C_VEL
LIN {X 0,Y 415.33,Z 698.609,A -85,B 0,C 180,E1 -10546.656,E2 -10546.656} C_VEL
LIN {X 0,Y 415.928,Z 685.91,A -85,B 0,C 180,E1 -10547.137,E2 -10547.137} C_VEL
LIN {X 0,Y 416.268,Z 672.593,A -85,B 0,C 180,E1 -10547.439,E2 -10547.439} C_VEL
LIN {X 0,Y 416.907,Z 597.409,A -85,B 0,C 180,E1 -10548.745,E2 -10548.745} C_VEL
LIN {X 0,Y 412.909,Z 572.92,A -85,B 0,C 180,E1 -10549.385,E2 -10549.385} C_VEL
LIN {X 0,Y 412.883,Z 571.797,A -85,B 0,C 180,E1 -10549.515,E2 -10549.515} C_VEL
LIN {X 0,Y 414.227,Z 553.166,A -85,B 0,C 180,E1 -10553.32,E2 -10553.32} C_VEL
LIN {X 0,Y 414.274,Z 548.527,A -85,B 0,C 180,E1 -10554.293,E2 -10554.293} C_VEL
LIN {X 0,Y 411.785,Z 535.561,A -85,B 0,C 180,E1 -10557.221,E2 -10557.221} C_VEL
LIN {X 0,Y 411.273,Z 533.29,A -85,B 0,C 180,E1 -10557.823,E2 -10557.823} C_VEL
LIN {X 0,Y 411.186,Z 533.267,A -85,B 0,C 180,E1 -10561.284,E2 -10561.284} C_VEL
LIN {X 0,Y 411.21,Z 533.266,A -85,B 0,C 180,E1 -10564.334,E2 -10564.334} C_VEL
LIN {X 0,Y 411.198,Z 533.267,A -85,B 0,C 180,E1 -10567.974,E2 -10567.974} C_VEL
LIN {X 0,Y 411.167,Z 533.267,A -85,B 0,C 180,E1 -10571.229,E2 -10571.229} C_VEL
LIN {X 0,Y 411.18,Z 533.266,A -85,B 0,C 180,E1 -10574.491,E2 -10574.491} C_VEL
LIN {X 0,Y 411.181,Z 533.268,A -85,B 0,C 180,E1 -10578.195,E2 -10578.195} C_VEL
LIN {X 0,Y 411.223,Z 533.259,A -85,B 0,C 180,E1 -10580.776,E2 -10580.776} C_VEL
LIN {X 0,Y 411.204,Z 533.264,A -85,B 0,C 180,E1 -10584.472,E2 -10584.472} C_VEL
LIN {X 0,Y 411.211,Z 533.264,A -85,B 0,C 180,E1 -10586.874,E2 -10586.874} C_VEL
LIN {X 0,Y 411.246,Z 533.505,A -85,B 0,C 180,E1 -10589.62,E2 -10589.62} C_VEL
LIN {X 0,Y 413.821,Z 542.38,A -85,B 0,C 180,E1 -10591.341,E2 -10591.341} C_VEL
LIN {X 0,Y 415.808,Z 552.122,A -85,B 0,C 180,E1 -10593.083,E2 -10593.083} C_VEL
LIN {X 0,Y 415.843,Z 557.399,A -85,B 0,C 180,E1 -10593.933,E2 -10593.933} C_VEL
LIN {X 0,Y 414.795,Z 577.297,A -85,B 0,C 180,E1 -10597.064,E2 -10597.064} C_VEL
LIN {X 0,Y 413.896,Z 596.967,A -85,B 0,C 180,E1 -10600.147,E2 -10600.147} C_VEL
LIN {X 0,Y 412.965,Z 619.471,A -85,B 0,C 180,E1 -10603.692,E2 -10603.692} C_VEL
LIN {X 0,Y 412.509,Z 631.848,A -85,B 0,C 180,E1 -10605.603,E2 -10605.603} C_VEL
LIN {X 0,Y 414.386,Z 646.628,A -85,B 0,C 180,E1 -10606.058,E2 -10606.058} C_VEL
LIN {X 0,Y 413.366,Z 704.464,A -85,B 0,C 180,E1 -10607.356,E2 -10607.356} C_VEL
LIN {X 0,Y 413.025,Z 714.153,A -85,B 0,C 180,E1 -10607.719,E2 -10607.719} C_VEL
LIN {X 0,Y 412.671,Z 724.405,A -85,B 0,C 180,E1 -10608.27,E2 -10608.27} C_VEL
LIN {X 0,Y 412.182,Z 734.997,A -85,B 0,C 180,E1 -10609.065,E2 -10609.065} C_VEL
LIN {X 0,Y 411.767,Z 743.848,A -85,B 0,C 180,E1 -10609.924,E2 -10609.924} C_VEL
LIN {X 0,Y 411.246,Z 751.864,A -85,B 0,C 180,E1 -10610.905,E2 -10610.905} C_VEL
LIN {X 0,Y 410.888,Z 758.232,A -85,B 0,C 180,E1 -10611.888,E2 -10611.888} C_VEL
LIN {X 0,Y 410.545,Z 764.631,A -85,B 0,C 180,E1 -10613.118,E2 -10613.118} C_VEL
LIN {X 0,Y 410.45,Z 768.715,A -85,B 0,C 180,E1 -10614.103,E2 -10614.103} C_VEL
LIN {X 0,Y 410.099,Z 773.44,A -85,B 0,C 180,E1 -10615.577,E2 -10615.577} C_VEL
LIN {X 0,Y 410.022,Z 776.534,A -85,B 0,C 180,E1 -10617.052,E2 -10617.052} C_VEL
LIN {X 0,Y 409.977,Z 777.872,A -85,B 0,C 180,E1 -10618.035,E2 -10618.035} C_VEL
LIN {X 0,Y 409.919,Z 778.633,A -85,B 0,C 180,E1 -10619.018,E2 -10619.018} C_VEL
LIN {X 0,Y 409.906,Z 778.827,A -85,B 0,C 180,E1 -10620,E2 -10620} C_VEL
LIN {X 0,Y 409.919,Z 778.439,A -85,B 0,C 180,E1 -10620.982,E2 -10620.982} C_VEL
LIN {X 0,Y 409.973,Z 777.448,A -85,B 0,C 180,E1 -10621.965,E2 -10621.965} C_VEL
LIN {X 0,Y 410.011,Z 774.782,A -85,B 0,C 180,E1 -10623.44,E2 -10623.44} C_VEL
LIN {X 0,Y 410.154,Z 770.713,A -85,B 0,C 180,E1 -10624.915,E2 -10624.915} C_VEL
LIN {X 0,Y 410.264,Z 765.813,A -85,B 0,C 180,E1 -10626.21,E2 -10626.21} C_VEL
LIN {X 0,Y 410.551,Z 759.997,A -85,B 0,C 180,E1 -10627.377,E2 -10627.377} C_VEL
LIN {X 0,Y 410.754,Z 753.926,A -85,B 0,C 180,E1 -10628.363,E2 -10628.363} C_VEL
LIN {X 0,Y 411.191,Z 745.493,A -85,B 0,C 180,E1 -10629.469,E2 -10629.469} C_VEL
LIN {X 0,Y 411.546,Z 737.014,A -85,B 0,C 180,E1 -10630.33,E2 -10630.33} C_VEL
LIN {X 0,Y 411.947,Z 727.779,A -85,B 0,C 180,E1 -10631.066,E2 -10631.066} C_VEL
LIN {X 0,Y 412.239,Z 717.744,A -85,B 0,C 180,E1 -10631.68,E2 -10631.68} C_VEL
LIN {X 0,Y 412.557,Z 706.542,A -85,B 0,C 180,E1 -10632.139,E2 -10632.139} C_VEL
LIN {X 0,Y 412.679,Z 695.766,A -85,B 0,C 180,E1 -10632.416,E2 -10632.416} C_VEL
LIN {X 0,Y 413.183,Z 645.17,A -85,B 0,C 180,E1 -10633.46,E2 -10633.46} C_VEL
LIN {X 0,Y 411.783,Z 631.415,A -85,B 0,C 180,E1 -10633.824,E2 -10633.824} C_VEL
LIN {X 0,Y 412.612,Z 609.241,A -85,B 0,C 180,E1 -10637.316,E2 -10637.316} C_VEL
LIN {X 0,Y 413.514,Z 586.648,A -85,B 0,C 180,E1 -10640.911,E2 -10640.911} C_VEL
LIN {X 0,Y 414.399,Z 567.146,A -85,B 0,C 180,E1 -10644.018,E2 -10644.018} C_VEL
LIN {X 0,Y 415.117,Z 552.519,A -85,B 0,C 180,E1 -10646.359,E2 -10646.359} C_VEL
LIN {X 0,Y 412.986,Z 541.429,A -85,B 0,C 180,E1 -10648.262,E2 -10648.262} C_VEL
LIN {X 0,Y 411.268,Z 533.37,A -85,B 0,C 180,E1 -10649.707,E2 -10649.707} C_VEL
LIN {X 0,Y 411.211,Z 533.262,A -85,B 0,C 180,E1 -10653.156,E2 -10653.156} C_VEL
LIN {X 0,Y 411.2,Z 533.267,A -85,B 0,C 180,E1 -10656.553,E2 -10656.553} C_VEL
LIN {X 0,Y 411.218,Z 533.257,A -85,B 0,C 180,E1 -10659.728,E2 -10659.728} C_VEL
LIN {X 0,Y 411.177,Z 533.239,A -85,B 0,C 180,E1 -10663.133,E2 -10663.133} C_VEL
LIN {X 0,Y 411.177,Z 533.262,A -85,B 0,C 180,E1 -10665.88,E2 -10665.88} C_VEL
LIN {X 0,Y 411.172,Z 533.257,A -85,B 0,C 180,E1 -10668.771,E2 -10668.771} C_VEL
LIN {X 0,Y 411.197,Z 533.255,A -85,B 0,C 180,E1 -10672.026,E2 -10672.026} C_VEL
LIN {X 0,Y 411.21,Z 533.253,A -85,B 0,C 180,E1 -10675.666,E2 -10675.666} C_VEL
LIN {X 0,Y 411.194,Z 533.263,A -85,B 0,C 180,E1 -10679.152,E2 -10679.152} C_VEL
LIN {X 0,Y 411.263,Z 533.26,A -85,B 0,C 180,E1 -10682.522,E2 -10682.522} C_VEL
LIN {X 0,Y 411.278,Z 533.362,A -85,B 0,C 180,E1 -10686.256,E2 -10686.256} C_VEL
LIN {X 0,Y 413.364,Z 544.707,A -85,B 0,C 180,E1 -10689.246,E2 -10689.246} C_VEL
LIN {X 0,Y 413.127,Z 550.758,A -85,B 0,C 180,E1 -10690.649,E2 -10690.649} C_VEL
LIN {X 0,Y 414.568,Z 557.857,A -85,B 0,C 180,E1 -10690.888,E2 -10690.888} C_VEL
LIN {X 0,Y 417.301,Z 572.09,A -85,B 0,C 180,E1 -10691.273,E2 -10691.273} C_VEL
LIN {X 0,Y 416.281,Z 656.855,A -85,B 0,C 180,E1 -10692.751,E2 -10692.751} C_VEL
LIN {X 0,Y 415.884,Z 669.605,A -85,B 0,C 180,E1 -10693.146,E2 -10693.146} C_VEL
LIN {X 0,Y 415.286,Z 683.168,A -85,B 0,C 180,E1 -10693.785,E2 -10693.785} C_VEL
LIN {X 0,Y 414.642,Z 694.528,A -85,B 0,C 180,E1 -10694.517,E2 -10694.517} C_VEL
LIN {X 0,Y 413.613,Z 699.763,A -85,B 0,C 180,E1 -10694.897,E2 -10694.897} C_VEL
LIN {X 0,Y 408.853,Z 711.095,A -85,B 0,C 180,E1 -10695.8,E2 -10695.8} C_VEL
LIN {X 0,Y 406.551,Z 717.189,A -85,B 0,C 180,E1 -10696.418,E2 -10696.418} C_VEL
LIN {X 0,Y 406.01,Z 720.118,A -85,B 0,C 180,E1 -10696.773,E2 -10696.773} C_VEL
LIN {X 0,Y 405.185,Z 728.713,A -85,B 0,C 180,E1 -10697.986,E2 -10697.986} C_VEL
LIN {X 0,Y 404.509,Z 737.338,A -85,B 0,C 180,E1 -10699.488,E2 -10699.488} C_VEL
LIN {X 0,Y 403.919,Z 744.212,A -85,B 0,C 180,E1 -10700.99,E2 -10700.99} C_VEL
LIN {X 0,Y 403.475,Z 749.718,A -85,B 0,C 180,E1 -10702.493,E2 -10702.493} C_VEL
LIN {X 0,Y 403.28,Z 754.034,A -85,B 0,C 180,E1 -10703.997,E2 -10703.997} C_VEL
LIN {X 0,Y 403.11,Z 756.317,A -85,B 0,C 180,E1 -10704.998,E2 -10704.998} C_VEL
LIN {X 0,Y 402.975,Z 758.177,A -85,B 0,C 180,E1 -10705.999,E2 -10705.999} C_VEL
LIN {X 0,Y 402.964,Z 759.576,A -85,B 0,C 180,E1 -10707,E2 -10707} C_VEL
LIN {X 0,Y 402.945,Z 760.572,A -85,B 0,C 180,E1 -10708,E2 -10708} C_VEL
LIN {X 0,Y 402.851,Z 761.423,A -85,B 0,C 180,E1 -10709.999,E2 -10709.999} C_VEL
LIN {X 0,Y 402.867,Z 761.236,A -85,B 0,C 180,E1 -10710.999,E2 -10710.999} C_VEL
LIN {X 0,Y 402.945,Z 760.651,A -85,B 0,C 180,E1 -10711.998,E2 -10711.998} C_VEL
LIN {X 0,Y 402.959,Z 759.688,A -85,B 0,C 180,E1 -10712.998,E2 -10712.998} C_VEL
LIN {X 0,Y 402.964,Z 758.335,A -85,B 0,C 180,E1 -10713.999,E2 -10713.999} C_VEL
LIN {X 0,Y 403.215,Z 755.466,A -85,B 0,C 180,E1 -10715.5,E2 -10715.5} C_VEL
LIN {X 0,Y 403.403,Z 751.58,A -85,B 0,C 180,E1 -10717.004,E2 -10717.004} C_VEL
LIN {X 0,Y 403.716,Z 746.571,A -85,B 0,C 180,E1 -10718.508,E2 -10718.508} C_VEL
LIN {X 0,Y 404.282,Z 740.261,A -85,B 0,C 180,E1 -10720.01,E2 -10720.01} C_VEL
LIN {X 0,Y 404.96,Z 732.359,A -85,B 0,C 180,E1 -10721.511,E2 -10721.511} C_VEL
LIN {X 0,Y 405.618,Z 724.305,A -85,B 0,C 180,E1 -10722.762,E2 -10722.762} C_VEL
LIN {X 0,Y 406.5,Z 714.47,A -85,B 0,C 180,E1 -10724.006,E2 -10724.006} C_VEL
LIN {X 0,Y 407.203,Z 703.419,A -85,B 0,C 180,E1 -10725.131,E2 -10725.131} C_VEL
LIN {X 0,Y 407.981,Z 692.572,A -85,B 0,C 180,E1 -10725.998,E2 -10725.998} C_VEL
LIN {X 0,Y 408.706,Z 680.583,A -85,B 0,C 180,E1 -10726.739,E2 -10726.739} C_VEL
LIN {X 0,Y 409.207,Z 668.308,A -85,B 0,C 180,E1 -10727.297,E2 -10727.297} C_VEL
LIN {X 0,Y 409.613,Z 655.674,A -85,B 0,C 180,E1 -10727.665,E2 -10727.665} C_VEL
LIN {X 0,Y 410.421,Z 571.685,A -85,B 0,C 180,E1 -10729.161,E2 -10729.161} C_VEL
LIN {X 0,Y 406.256,Z 551.18,A -85,B 0,C 180,E1 -10729.772,E2 -10729.772} C_VEL
LIN {X 0,Y 406.319,Z 548.894,A -85,B 0,C 180,E1 -10730.238,E2 -10730.238} C_VEL
LIN {X 0,Y 406.192,Z 544.632,A -85,B 0,C 180,E1 -10731.305,E2 -10731.305} C_VEL
LIN {X 0,Y 404.227,Z 534.223,A -85,B 0,C 180,E1 -10734.114,E2 -10734.114} C_VEL
LIN {X 0,Y 404.225,Z 534.136,A -85,B 0,C 180,E1 -10737.537,E2 -10737.537} C_VEL
LIN {X 0,Y 404.144,Z 534.137,A -85,B 0,C 180,E1 -10740.284,E2 -10740.284} C_VEL
LIN {X 0,Y 404.143,Z 534.145,A -85,B 0,C 180,E1 -10743.811,E2 -10743.811} C_VEL
LIN {X 0,Y 404.137,Z 534.139,A -85,B 0,C 180,E1 -10746.875,E2 -10746.875} C_VEL
LIN {X 0,Y 404.156,Z 534.134,A -85,B 0,C 180,E1 -10750.081,E2 -10750.081} C_VEL
LIN {X 0,Y 404.153,Z 534.143,A -85,B 0,C 180,E1 -10753.083,E2 -10753.083} C_VEL
LIN {X 0,Y 404.144,Z 534.139,A -85,B 0,C 180,E1 -10755.925,E2 -10755.925} C_VEL
LIN {X 0,Y 404.147,Z 534.14,A -85,B 0,C 180,E1 -10758.638,E2 -10758.638} C_VEL
LIN {X 0,Y 404.157,Z 534.125,A -85,B 0,C 180,E1 -10761.49,E2 -10761.49} C_VEL
LIN {X 0,Y 404.182,Z 534.137,A -85,B 0,C 180,E1 -10764.983,E2 -10764.983} C_VEL
LIN {X 0,Y 404.14,Z 534.138,A -85,B 0,C 180,E1 -10768.553,E2 -10768.553} C_VEL
LIN {X 0,Y 404.192,Z 534.128,A -85,B 0,C 180,E1 -10772,E2 -10772} C_VEL
LIN {X 0,Y 404.171,Z 534.142,A -85,B 0,C 180,E1 -10775.334,E2 -10775.334} C_VEL
LIN {X 0,Y 404.132,Z 534.135,A -85,B 0,C 180,E1 -10778.58,E2 -10778.58} C_VEL
LIN {X 0,Y 404.203,Z 534.133,A -85,B 0,C 180,E1 -10781.761,E2 -10781.761} C_VEL
LIN {X 0,Y 404.199,Z 534.127,A -85,B 0,C 180,E1 -10784.882,E2 -10784.882} C_VEL
LIN {X 0,Y 404.249,Z 534.126,A -85,B 0,C 180,E1 -10787.958,E2 -10787.958} C_VEL
LIN {X 0,Y 404.425,Z 534.105,A -85,B 0,C 180,E1 -10792.099,E2 -10792.099} C_VEL
LIN {X 0,Y 404.416,Z 534.107,A -85,B 0,C 180,E1 -10794.015,E2 -10794.015} C_VEL
LIN {X 0,Y 404.475,Z 534.098,A -85,B 0,C 180,E1 -10798.008,E2 -10798.008} C_VEL
LIN {X 0,Y 404.606,Z 534.085,A -85,B 0,C 180,E1 -10800,E2 -10800} C_VEL
LIN {X 0,Y 404.417,Z 534.102,A -85,B 0,C 180,E1 -10802.988,E2 -10802.988} C_VEL
LIN {X 0,Y 404.427,Z 534.107,A -85,B 0,C 180,E1 -10805.985,E2 -10805.985} C_VEL
LIN {X 0,Y 404.415,Z 534.106,A -85,B 0,C 180,E1 -10807.991,E2 -10807.991} C_VEL
LIN {X 0,Y 404.262,Z 534.127,A -85,B 0,C 180,E1 -10812.041,E2 -10812.041} C_VEL
LIN {X 0,Y 404.2,Z 534.133,A -85,B 0,C 180,E1 -10815.118,E2 -10815.118} C_VEL
LIN {X 0,Y 404.206,Z 534.133,A -85,B 0,C 180,E1 -10818.238,E2 -10818.238} C_VEL
LIN {X 0,Y 404.156,Z 534.138,A -85,B 0,C 180,E1 -10821.418,E2 -10821.418} C_VEL
LIN {X 0,Y 404.17,Z 534.137,A -85,B 0,C 180,E1 -10824.666,E2 -10824.666} C_VEL
LIN {X 0,Y 404.188,Z 534.138,A -85,B 0,C 180,E1 -10828,E2 -10828} C_VEL
LIN {X 0,Y 404.135,Z 534.142,A -85,B 0,C 180,E1 -10831.559,E2 -10831.559} C_VEL
LIN {X 0,Y 404.179,Z 534.133,A -85,B 0,C 180,E1 -10835.017,E2 -10835.017} C_VEL
LIN {X 0,Y 404.154,Z 534.138,A -85,B 0,C 180,E1 -10838.757,E2 -10838.757} C_VEL
LIN {X 0,Y 404.118,Z 534.14,A -85,B 0,C 180,E1 -10841.601,E2 -10841.601} C_VEL
LIN {X 0,Y 404.15,Z 534.14,A -85,B 0,C 180,E1 -10844.524,E2 -10844.524} C_VEL
LIN {X 0,Y 404.203,Z 534.129,A -85,B 0,C 180,E1 -10847.306,E2 -10847.306} C_VEL
LIN {X 0,Y 404.165,Z 534.136,A -85,B 0,C 180,E1 -10849.956,E2 -10849.956} C_VEL
LIN {X 0,Y 404.137,Z 534.129,A -85,B 0,C 180,E1 -10853.125,E2 -10853.125} C_VEL
LIN {X 0,Y 404.142,Z 534.133,A -85,B 0,C 180,E1 -10856.189,E2 -10856.189} C_VEL
LIN {X 0,Y 404.143,Z 534.093,A -85,B 0,C 180,E1 -10859.716,E2 -10859.716} C_VEL
LIN {X 0,Y 404.267,Z 534.351,A -85,B 0,C 180,E1 -10861.972,E2 -10861.972} C_VEL
LIN {X 0,Y 406.854,Z 547.107,A -85,B 0,C 180,E1 -10864.964,E2 -10864.964} C_VEL
LIN {X 0,Y 407.442,Z 552.195,A -85,B 0,C 180,E1 -10866.093,E2 -10866.093} C_VEL
LIN {X 0,Y 406.221,Z 568.069,A -85,B 0,C 180,E1 -10869.411,E2 -10869.411} C_VEL
LIN {X 0,Y 405.96,Z 572.311,A -85,B 0,C 180,E1 -10870.239,E2 -10870.239} C_VEL
LIN {X 0,Y 410.326,Z 599.278,A -85,B 0,C 180,E1 -10870.974,E2 -10870.974} C_VEL
LIN {X 0,Y 409.353,Z 680.376,A -85,B 0,C 180,E1 -10872.42,E2 -10872.42} C_VEL
LIN {X 0,Y 408.744,Z 693.599,A -85,B 0,C 180,E1 -10872.844,E2 -10872.844} C_VEL
LIN {X 0,Y 408.147,Z 705.746,A -85,B 0,C 180,E1 -10873.431,E2 -10873.431} C_VEL
LIN {X 0,Y 407.332,Z 718.011,A -85,B 0,C 180,E1 -10874.233,E2 -10874.233} C_VEL
LIN {X 0,Y 406.429,Z 729.86,A -85,B 0,C 180,E1 -10875.25,E2 -10875.25} C_VEL
LIN {X 0,Y 405.657,Z 740.039,A -85,B 0,C 180,E1 -10876.347,E2 -10876.347} C_VEL
LIN {X 0,Y 405,Z 748.578,A -85,B 0,C 180,E1 -10877.473,E2 -10877.473} C_VEL
LIN {X 0,Y 404.323,Z 756.453,A -85,B 0,C 180,E1 -10878.724,E2 -10878.724} C_VEL
LIN {X 0,Y 403.722,Z 764.149,A -85,B 0,C 180,E1 -10880.229,E2 -10880.229} C_VEL
LIN {X 0,Y 403.287,Z 771.245,A -85,B 0,C 180,E1 -10881.987,E2 -10881.987} C_VEL
LIN {X 0,Y 402.957,Z 776.787,A -85,B 0,C 180,E1 -10883.796,E2 -10883.796} C_VEL
LIN {X 0,Y 402.937,Z 779.582,A -85,B 0,C 180,E1 -10884.998,E2 -10884.998} C_VEL
LIN {X 0,Y 402.855,Z 781.444,A -85,B 0,C 180,E1 -10885.999,E2 -10885.999} C_VEL
LIN {X 0,Y 402.864,Z 783.836,A -85,B 0,C 180,E1 -10888.001,E2 -10888.001} C_VEL
LIN {X 0,Y 402.851,Z 785.021,A -85,B 0,C 180,E1 -10890.001,E2 -10890.001} C_VEL
LIN {X 0,Y 402.862,Z 784.876,A -85,B 0,C 180,E1 -10891,E2 -10891} C_VEL
LIN {X 0,Y 402.864,Z 784.148,A -85,B 0,C 180,E1 -10892,E2 -10892} C_VEL
LIN {X 0,Y 402.856,Z 781.429,A -85,B 0,C 180,E1 -10894.002,E2 -10894.002} C_VEL
LIN {X 0,Y 402.928,Z 778.492,A -85,B 0,C 180,E1 -10895.506,E2 -10895.506} C_VEL
LIN {X 0,Y 403.083,Z 774.516,A -85,B 0,C 180,E1 -10897.011,E2 -10897.011} C_VEL
LIN {X 0,Y 403.432,Z 768.398,A -85,B 0,C 180,E1 -10898.769,E2 -10898.769} C_VEL
LIN {X 0,Y 403.936,Z 761.717,A -85,B 0,C 180,E1 -10900.274,E2 -10900.274} C_VEL
LIN {X 0,Y 404.568,Z 753.429,A -85,B 0,C 180,E1 -10901.779,E2 -10901.779} C_VEL
LIN {X 0,Y 405.302,Z 744.936,A -85,B 0,C 180,E1 -10903.029,E2 -10903.029} C_VEL
LIN {X 0,Y 406.021,Z 734.939,A -85,B 0,C 180,E1 -10904.226,E2 -10904.226} C_VEL
LIN {X 0,Y 406.848,Z 724.055,A -85,B 0,C 180,E1 -10905.275,E2 -10905.275} C_VEL
LIN {X 0,Y 407.678,Z 712.68,A -85,B 0,C 180,E1 -10906.14,E2 -10906.14} C_VEL
LIN {X 0,Y 408.421,Z 701.003,A -85,B 0,C 180,E1 -10906.817,E2 -10906.817} C_VEL
LIN {X 0,Y 409.033,Z 688.447,A -85,B 0,C 180,E1 -10907.338,E2 -10907.338} C_VEL
LIN {X 0,Y 409.433,Z 675.697,A -85,B 0,C 180,E1 -10907.675,E2 -10907.675} C_VEL
LIN {X 0,Y 410.208,Z 598.431,A -85,B 0,C 180,E1 -10909.04,E2 -10909.04} C_VEL
LIN {X 0,Y 406.001,Z 572.7,A -85,B 0,C 180,E1 -10909.728,E2 -10909.728} C_VEL
LIN {X 0,Y 406.023,Z 570.911,A -85,B 0,C 180,E1 -10909.991,E2 -10909.991} C_VEL
LIN {X 0,Y 407.399,Z 552.864,A -85,B 0,C 180,E1 -10913.758,E2 -10913.758} C_VEL
LIN {X 0,Y 407.284,Z 549.594,A -85,B 0,C 180,E1 -10914.466,E2 -10914.466} C_VEL
LIN {X 0,Y 404.985,Z 537.634,A -85,B 0,C 180,E1 -10917.216,E2 -10917.216} C_VEL
LIN {X 0,Y 404.238,Z 534.186,A -85,B 0,C 180,E1 -10918.103,E2 -10918.103} C_VEL
LIN {X 0,Y 404.143,Z 534.145,A -85,B 0,C 180,E1 -10921.558,E2 -10921.558} C_VEL
LIN {X 0,Y 404.189,Z 534.136,A -85,B 0,C 180,E1 -10925.017,E2 -10925.017} C_VEL
LIN {X 0,Y 404.158,Z 534.139,A -85,B 0,C 180,E1 -10928.757,E2 -10928.757} C_VEL
LIN {X 0,Y 404.127,Z 534.146,A -85,B 0,C 180,E1 -10931.6,E2 -10931.6} C_VEL
LIN {X 0,Y 404.149,Z 534.141,A -85,B 0,C 180,E1 -10934.522,E2 -10934.522} C_VEL
LIN {X 0,Y 404.14,Z 534.145,A -85,B 0,C 180,E1 -10937.296,E2 -10937.296} C_VEL
LIN {X 0,Y 404.173,Z 534.141,A -85,B 0,C 180,E1 -10939.956,E2 -10939.956} C_VEL
LIN {X 0,Y 404.144,Z 534.145,A -85,B 0,C 180,E1 -10943.125,E2 -10943.125} C_VEL
LIN {X 0,Y 404.149,Z 534.144,A -85,B 0,C 180,E1 -10946.188,E2 -10946.188} C_VEL
LIN {X 0,Y 404.198,Z 534.327,A -85,B 0,C 180,E1 -10949.032,E2 -10949.032} C_VEL
LIN {X 0,Y 407.493,Z 545.706,A -85,B 0,C 180,E1 -10951.315,E2 -10951.315} C_VEL
LIN {X 0,Y 409.24,Z 554.475,A -85,B 0,C 180,E1 -10952.918,E2 -10952.918} C_VEL
LIN {X 0,Y 409.191,Z 559.588,A -85,B 0,C 180,E1 -10953.751,E2 -10953.751} C_VEL
LIN {X 0,Y 408.037,Z 579.496,A -85,B 0,C 180,E1 -10956.931,E2 -10956.931} C_VEL
LIN {X 0,Y 407.143,Z 597.547,A -85,B 0,C 180,E1 -10959.804,E2 -10959.804} C_VEL
LIN {X 0,Y 406.126,Z 620.096,A -85,B 0,C 180,E1 -10963.409,E2 -10963.409} C_VEL
LIN {X 0,Y 405.681,Z 631.898,A -85,B 0,C 180,E1 -10965.256,E2 -10965.256} C_VEL
LIN {X 0,Y 407.665,Z 647.205,A -85,B 0,C 180,E1 -10965.753,E2 -10965.753} C_VEL
LIN {X 0,Y 406.555,Z 704.635,A -85,B 0,C 180,E1 -10967.077,E2 -10967.077} C_VEL
LIN {X 0,Y 406.216,Z 714.264,A -85,B 0,C 180,E1 -10967.447,E2 -10967.447} C_VEL
LIN {X 0,Y 405.829,Z 724.488,A -85,B 0,C 180,E1 -10968.006,E2 -10968.006} C_VEL
LIN {X 0,Y 405.343,Z 734.324,A -85,B 0,C 180,E1 -10968.752,E2 -10968.752} C_VEL
LIN {X 0,Y 404.951,Z 742.088,A -85,B 0,C 180,E1 -10969.5,E2 -10969.5} C_VEL
LIN {X 0,Y 404.417,Z 750.477,A -85,B 0,C 180,E1 -10970.497,E2 -10970.497} C_VEL
LIN {X 0,Y 403.859,Z 758.569,A -85,B 0,C 180,E1 -10971.746,E2 -10971.746} C_VEL
LIN {X 0,Y 403.616,Z 763.765,A -85,B 0,C 180,E1 -10972.748,E2 -10972.748} C_VEL
LIN {X 0,Y 403.408,Z 768.983,A -85,B 0,C 180,E1 -10974,E2 -10974} C_VEL
LIN {X 0,Y 403.03,Z 773.632,A -85,B 0,C 180,E1 -10975.499,E2 -10975.499} C_VEL
LIN {X 0,Y 402.926,Z 776.693,A -85,B 0,C 180,E1 -10977.001,E2 -10977.001} C_VEL
LIN {X 0,Y 402.893,Z 777.992,A -85,B 0,C 180,E1 -10978.001,E2 -10978.001} C_VEL
LIN {X 0,Y 402.847,Z 778.713,A -85,B 0,C 180,E1 -10979,E2 -10979} C_VEL
LIN {X 0,Y 402.832,Z 778.862,A -85,B 0,C 180,E1 -10980,E2 -10980} C_VEL
LIN {X 0,Y 402.848,Z 778.435,A -85,B 0,C 180,E1 -10981,E2 -10981} C_VEL
LIN {X 0,Y 402.872,Z 777.412,A -85,B 0,C 180,E1 -10981.999,E2 -10981.999} C_VEL
LIN {X 0,Y 402.915,Z 774.665,A -85,B 0,C 180,E1 -10983.5,E2 -10983.5} C_VEL
LIN {X 0,Y 403.07,Z 770.538,A -85,B 0,C 180,E1 -10985.002,E2 -10985.002} C_VEL
LIN {X 0,Y 403.163,Z 766.184,A -85,B 0,C 180,E1 -10986.17,E2 -10986.17} C_VEL
LIN {X 0,Y 403.502,Z 759.615,A -85,B 0,C 180,E1 -10987.506,E2 -10987.506} C_VEL
LIN {X 0,Y 403.712,Z 753.457,A -85,B 0,C 180,E1 -10988.509,E2 -10988.509} C_VEL
LIN {X 0,Y 404.161,Z 744.864,A -85,B 0,C 180,E1 -10989.635,E2 -10989.635} C_VEL
LIN {X 0,Y 404.52,Z 736.176,A -85,B 0,C 180,E1 -10990.511,E2 -10990.511} C_VEL
LIN {X 0,Y 404.883,Z 728.483,A -85,B 0,C 180,E1 -10991.134,E2 -10991.134} C_VEL
LIN {X 0,Y 405.173,Z 718.647,A -85,B 0,C 180,E1 -10991.76,E2 -10991.76} C_VEL
LIN {X 0,Y 405.536,Z 707.204,A -85,B 0,C 180,E1 -10992.257,E2 -10992.257} C_VEL
LIN {X 0,Y 405.679,Z 695.436,A -85,B 0,C 180,E1 -10992.57,E2 -10992.57} C_VEL
LIN {X 0,Y 406.292,Z 646.443,A -85,B 0,C 180,E1 -10993.607,E2 -10993.607} C_VEL
LIN {X 0,Y 404.77,Z 631.545,A -85,B 0,C 180,E1 -10993.992,E2 -10993.992} C_VEL
LIN {X 0,Y 405.617,Z 609.616,A -85,B 0,C 180,E1 -10997.482,E2 -10997.482} C_VEL
LIN {X 0,Y 406.513,Z 587.738,A -85,B 0,C 180,E1 -11000.999,E2 -11000.999} C_VEL
LIN {X 0,Y 407.462,Z 567.528,A -85,B 0,C 180,E1 -11004.256,E2 -11004.256} C_VEL
LIN {X 0,Y 408.078,Z 553.058,A -85,B 0,C 180,E1 -11006.601,E2 -11006.601} C_VEL
LIN {X 0,Y 404.975,Z 537.712,A -85,B 0,C 180,E1 -11009.279,E2 -11009.279} C_VEL
LIN {X 0,Y 404.211,Z 534.245,A -85,B 0,C 180,E1 -11009.935,E2 -11009.935} C_VEL
LIN {X 0,Y 404.15,Z 534.143,A -85,B 0,C 180,E1 -11013.812,E2 -11013.812} C_VEL
LIN {X 0,Y 404.144,Z 534.143,A -85,B 0,C 180,E1 -11016.875,E2 -11016.875} C_VEL
LIN {X 0,Y 404.152,Z 534.138,A -85,B 0,C 180,E1 -11020.08,E2 -11020.08} C_VEL
LIN {X 0,Y 404.157,Z 534.112,A -85,B 0,C 180,E1 -11023.083,E2 -11023.083} C_VEL
LIN {X 0,Y 404.157,Z 534.136,A -85,B 0,C 180,E1 -11025.926,E2 -11025.926} C_VEL
LIN {X 0,Y 404.128,Z 534.136,A -85,B 0,C 180,E1 -11028.635,E2 -11028.635} C_VEL
LIN {X 0,Y 404.156,Z 534.13,A -85,B 0,C 180,E1 -11031.492,E2 -11031.492} C_VEL
LIN {X 0,Y 404.189,Z 534.129,A -85,B 0,C 180,E1 -11034.984,E2 -11034.984} C_VEL
LIN {X 0,Y 404.147,Z 534.14,A -85,B 0,C 180,E1 -11038.553,E2 -11038.553} C_VEL
LIN {X 0,Y 404.2,Z 534.135,A -85,B 0,C 180,E1 -11042,E2 -11042} C_VEL
LIN {X 0,Y 404.186,Z 534.129,A -85,B 0,C 180,E1 -11045.334,E2 -11045.334} C_VEL
LIN {X 0,Y 404.243,Z 534.295,A -85,B 0,C 180,E1 -11046.021,E2 -11046.021} C_VEL
LIN {X 0,Y 406.383,Z 545.607,A -85,B 0,C 180,E1 -11049.048,E2 -11049.048} C_VEL
LIN {X 0,Y 406.244,Z 550.962,A -85,B 0,C 180,E1 -11050.308,E2 -11050.308} C_VEL
LIN {X 0,Y 407.694,Z 558.164,A -85,B 0,C 180,E1 -11050.554,E2 -11050.554} C_VEL
LIN {X 0,Y 410.584,Z 572.675,A -85,B 0,C 180,E1 -11050.962,E2 -11050.962} C_VEL
LIN {X 0,Y 409.507,Z 657.079,A -85,B 0,C 180,E1 -11052.457,E2 -11052.457} C_VEL
LIN {X 0,Y 409.079,Z 670.582,A -85,B 0,C 180,E1 -11052.889,E2 -11052.889} C_VEL
LIN {X 0,Y 408.485,Z 683.38,A -85,B 0,C 180,E1 -11053.507,E2 -11053.507} C_VEL
